LIN {X 0,Y 411.178,Z 190.084,A -85,B 0,C 180,E1 -10484.491,E2 -10484.491} C_VEL
LIN {X 0,Y 411.179,Z 190.083,A -85,B 0,C 180,E1 -10488.195,E2 -10488.195} C_VEL
LIN {X 0,Y 411.222,Z 190.077,A -85,B 0,C 180,E1 -10490.776,E2 -10490.776} C_VEL
LIN {X 0,Y 411.215,Z 190.215,A -85,B 0,C 180,E1 -10492.954,E2 -10492.954} C_VEL
LIN {X 0,Y 412.247,Z 195.412,A -85,B 0,C 180,E1 -10495.765,E2 -10495.765} C_VEL
LIN {X 0,Y 413.023,Z 200.45,A -85,B 0,C 180,E1 -10498.299,E2 -10498.299} C_VEL
LIN {X 0,Y 412.701,Z 205.041,A -85,B 0,C 180,E1 -10500.406,E2 -10500.406} C_VEL
LIN {X 0,Y 411.967,Z 212.522,A -85,B 0,C 180,E1 -10503.67,E2 -10503.67} C_VEL
LIN {X 0,Y 411.402,Z 220.138,A -85,B 0,C 180,E1 -10506.864,E2 -10506.864} C_VEL
LIN {X 0,Y 410.884,Z 229.318,A -85,B 0,C 180,E1 -10510.596,E2 -10510.596} C_VEL
LIN {X 0,Y 410.423,Z 239.572,A -85,B 0,C 180,E1 -10514.608,E2 -10514.608} C_VEL
LIN {X 0,Y 410.27,Z 243.414,A -85,B 0,C 180,E1 -10516.093,E2 -10516.093} C_VEL
LIN {X 0,Y 411.974,Z 256.351,A -85,B 0,C 180,E1 -10516.662,E2 -10516.662} C_VEL
LIN {X 0,Y 412.639,Z 265.647,A -85,B 0,C 180,E1 -10517.208,E2 -10517.208} C_VEL
LIN {X 0,Y 412.418,Z 274.261,A -85,B 0,C 180,E1 -10517.826,E2 -10517.826} C_VEL
LIN {X 0,Y 411.868,Z 282.527,A -85,B 0,C 180,E1 -10518.559,E2 -10518.559} C_VEL
LIN {X 0,Y 411.453,Z 290.378,A -85,B 0,C 180,E1 -10519.419,E2 -10519.419} C_VEL
LIN {X 0,Y 410.999,Z 297.735,A -85,B 0,C 180,E1 -10520.403,E2 -10520.403} C_VEL
LIN {X 0,Y 410.581,Z 305.203,A -85,B 0,C 180,E1 -10521.634,E2 -10521.634} C_VEL
LIN {X 0,Y 410.3,Z 311.045,A -85,B 0,C 180,E1 -10522.866,E2 -10522.866} C_VEL
LIN {X 0,Y 410.073,Z 315.663,A -85,B 0,C 180,E1 -10524.098,E2 -10524.098} C_VEL
LIN {X 0,Y 410.069,Z 318.666,A -85,B 0,C 180,E1 -10525.084,E2 -10525.084} C_VEL
LIN {X 0,Y 409.971,Z 321.016,A -85,B 0,C 180,E1 -10526.068,E2 -10526.068} C_VEL
LIN {X 0,Y 409.986,Z 322.747,A -85,B 0,C 180,E1 -10527.052,E2 -10527.052} C_VEL
LIN {X 0,Y 410.02,Z 323.966,A -85,B 0,C 180,E1 -10528.036,E2 -10528.036} C_VEL
LIN {X 0,Y 409.979,Z 324.696,A -85,B 0,C 180,E1 -10529.018,E2 -10529.018} C_VEL
LIN {X 0,Y 409.975,Z 324.952,A -85,B 0,C 180,E1 -10530,E2 -10530} C_VEL
LIN {X 0,Y 409.979,Z 324.652,A -85,B 0,C 180,E1 -10530.982,E2 -10530.982} C_VEL
LIN {X 0,Y 410.022,Z 323.785,A -85,B 0,C 180,E1 -10531.965,E2 -10531.965} C_VEL
LIN {X 0,Y 410.003,Z 322.422,A -85,B 0,C 180,E1 -10532.948,E2 -10532.948} C_VEL
LIN {X 0,Y 410.019,Z 319.386,A -85,B 0,C 180,E1 -10534.424,E2 -10534.424} C_VEL
LIN {X 0,Y 410.058,Z 315.019,A -85,B 0,C 180,E1 -10535.903,E2 -10535.903} C_VEL
LIN {X 0,Y 410.301,Z 310.119,A -85,B 0,C 180,E1 -10537.134,E2 -10537.134} C_VEL
LIN {X 0,Y 410.535,Z 303.893,A -85,B 0,C 180,E1 -10538.367,E2 -10538.367} C_VEL
LIN {X 0,Y 410.85,Z 297.806,A -85,B 0,C 180,E1 -10539.353,E2 -10539.353} C_VEL
LIN {X 0,Y 411.256,Z 290.392,A -85,B 0,C 180,E1 -10540.337,E2 -10540.337} C_VEL
LIN {X 0,Y 411.655,Z 282.441,A -85,B 0,C 180,E1 -10541.198,E2 -10541.198} C_VEL
LIN {X 0,Y 412.183,Z 272.525,A -85,B 0,C 180,E1 -10542.056,E2 -10542.056} C_VEL
LIN {X 0,Y 412.205,Z 264.215,A -85,B 0,C 180,E1 -10542.618,E2 -10542.618} C_VEL
LIN {X 0,Y 411.237,Z 253.02,A -85,B 0,C 180,E1 -10543.199,E2 -10543.199} C_VEL
LIN {X 0,Y 410.259,Z 244.088,A -85,B 0,C 180,E1 -10543.564,E2 -10543.564} C_VEL
LIN {X 0,Y 410.555,Z 235.397,A -85,B 0,C 180,E1 -10546.919,E2 -10546.919} C_VEL
LIN {X 0,Y 410.898,Z 227.517,A -85,B 0,C 180,E1 -10550.004,E2 -10550.004} C_VEL
LIN {X 0,Y 411.352,Z 219.645,A -85,B 0,C 180,E1 -10553.139,E2 -10553.139} C_VEL
LIN {X 0,Y 411.895,Z 211.789,A -85,B 0,C 180,E1 -10556.336,E2 -10556.336} C_VEL
LIN {X 0,Y 412.58,Z 203.75,A -85,B 0,C 180,E1 -10559.686,E2 -10559.686} C_VEL
LIN {X 0,Y 412.789,Z 199.19,A -85,B 0,C 180,E1 -10561.648,E2 -10561.648} C_VEL
LIN {X 0,Y 411.614,Z 192.001,A -85,B 0,C 180,E1 -10564.958,E2 -10564.958} C_VEL
LIN {X 0,Y 411.229,Z 190.075,A -85,B 0,C 180,E1 -10565.978,E2 -10565.978} C_VEL
LIN {X 0,Y 411.215,Z 190.075,A -85,B 0,C 180,E1 -10569.727,E2 -10569.727} C_VEL
LIN {X 0,Y 411.177,Z 190.079,A -85,B 0,C 180,E1 -10573.134,E2 -10573.134} C_VEL
LIN {X 0,Y 411.171,Z 190.081,A -85,B 0,C 180,E1 -10575.881,E2 -10575.881} C_VEL
LIN {X 0,Y 411.162,Z 190.083,A -85,B 0,C 180,E1 -10578.773,E2 -10578.773} C_VEL
LIN {X 0,Y 411.191,Z 190.081,A -85,B 0,C 180,E1 -10582.025,E2 -10582.025} C_VEL
LIN {X 0,Y 411.21,Z 190.076,A -85,B 0,C 180,E1 -10585.666,E2 -10585.666} C_VEL
LIN {X 0,Y 411.194,Z 190.076,A -85,B 0,C 180,E1 -10589.152,E2 -10589.152} C_VEL
LIN {X 0,Y 411.263,Z 190.068,A -85,B 0,C 180,E1 -10592.522,E2 -10592.522} C_VEL
LIN {X 0,Y 411.224,Z 190.076,A -85,B 0,C 180,E1 -10595.784,E2 -10595.784} C_VEL
LIN {X 0,Y 411.201,Z 190.076,A -85,B 0,C 180,E1 -10598.965,E2 -10598.965} C_VEL
LIN {X 0,Y 411.255,Z 190.071,A -85,B 0,C 180,E1 -10602.084,E2 -10602.084} C_VEL
LIN {X 0,Y 411.265,Z 190.07,A -85,B 0,C 180,E1 -10605.147,E2 -10605.147} C_VEL
LIN {X 0,Y 411.287,Z 190.066,A -85,B 0,C 180,E1 -10608.167,E2 -10608.167} C_VEL
LIN {X 0,Y 411.442,Z 190.046,A -85,B 0,C 180,E1 -10612.191,E2 -10612.191} C_VEL
LIN {X 0,Y 411.47,Z 190.042,A -85,B 0,C 180,E1 -10614.117,E2 -10614.117} C_VEL
LIN {X 0,Y 411.514,Z 190.036,A -85,B 0,C 180,E1 -10618.042,E2 -10618.042} C_VEL
LIN {X 0,Y 411.642,Z 190.021,A -85,B 0,C 180,E1 -10619.999,E2 -10619.999} C_VEL
LIN {X 0,Y 411.46,Z 190.047,A -85,B 0,C 180,E1 -10622.936,E2 -10622.936} C_VEL
LIN {X 0,Y 411.435,Z 190.048,A -85,B 0,C 180,E1 -10626.651,E2 -10626.651} C_VEL
LIN {X 0,Y 411.321,Z 190.064,A -85,B 0,C 180,E1 -10628.845,E2 -10628.845} C_VEL
LIN {X 0,Y 411.285,Z 190.065,A -85,B 0,C 180,E1 -10631.832,E2 -10631.832} C_VEL
LIN {X 0,Y 411.262,Z 190.071,A -85,B 0,C 180,E1 -10634.852,E2 -10634.852} C_VEL
LIN {X 0,Y 411.247,Z 190.07,A -85,B 0,C 180,E1 -10637.914,E2 -10637.914} C_VEL
LIN {X 0,Y 411.197,Z 190.078,A -85,B 0,C 180,E1 -10641.033,E2 -10641.033} C_VEL
LIN {X 0,Y 411.219,Z 190.075,A -85,B 0,C 180,E1 -10644.215,E2 -10644.215} C_VEL
LIN {X 0,Y 411.258,Z 190.068,A -85,B 0,C 180,E1 -10647.476,E2 -10647.476} C_VEL
LIN {X 0,Y 411.188,Z 190.079,A -85,B 0,C 180,E1 -10650.846,E2 -10650.846} C_VEL
LIN {X 0,Y 411.204,Z 190.079,A -85,B 0,C 180,E1 -10654.332,E2 -10654.332} C_VEL
LIN {X 0,Y 411.196,Z 190.079,A -85,B 0,C 180,E1 -10657.972,E2 -10657.972} C_VEL
LIN {X 0,Y 411.16,Z 190.081,A -85,B 0,C 180,E1 -10661.227,E2 -10661.227} C_VEL
LIN {X 0,Y 411.171,Z 190.081,A -85,B 0,C 180,E1 -10664.489,E2 -10664.489} C_VEL
LIN {X 0,Y 411.172,Z 190.082,A -85,B 0,C 180,E1 -10668.194,E2 -10668.194} C_VEL
LIN {X 0,Y 411.213,Z 190.074,A -85,B 0,C 180,E1 -10670.775,E2 -10670.775} C_VEL
LIN {X 0,Y 411.194,Z 190.077,A -85,B 0,C 180,E1 -10674.47,E2 -10674.47} C_VEL
LIN {X 0,Y 411.201,Z 190.076,A -85,B 0,C 180,E1 -10676.872,E2 -10676.872} C_VEL
LIN {X 0,Y 411.234,Z 190.071,A -85,B 0,C 180,E1 -10680.641,E2 -10680.641} C_VEL
LIN {X 0,Y 411.231,Z 190.075,A -85,B 0,C 180,E1 -10683.618,E2 -10683.618} C_VEL
LIN {X 0,Y 411.196,Z 190.078,A -85,B 0,C 180,E1 -10686.852,E2 -10686.852} C_VEL
LIN {X 0,Y 411.207,Z 190.076,A -85,B 0,C 180,E1 -10690.05,E2 -10690.05} C_VEL
LIN {X 0,Y 411.255,Z 190.073,A -85,B 0,C 180,E1 -10693.131,E2 -10693.131} C_VEL
LIN {X 0,Y 411.306,Z 190.066,A -85,B 0,C 180,E1 -10696.89,E2 -10696.89} C_VEL
LIN {X 0,Y 411.3,Z 190.062,A -85,B 0,C 180,E1 -10700.161,E2 -10700.161} C_VEL
LIN {X 0,Y 411.452,Z 190.048,A -85,B 0,C 180,E1 -10703.133,E2 -10703.133} C_VEL
LIN {X 0,Y 411.302,Z 190.066,A -85,B 0,C 180,E1 -10705.099,E2 -10705.099} C_VEL
LIN {X 0,Y 411.502,Z 190.038,A -85,B 0,C 180,E1 -10708.042,E2 -10708.042} C_VEL
LIN {X 0,Y 411.632,Z 190.023,A -85,B 0,C 180,E1 -10710,E2 -10710} C_VEL
LIN {X 0,Y 411.458,Z 190.047,A -85,B 0,C 180,E1 -10712.937,E2 -10712.937} C_VEL
LIN {X 0,Y 411.452,Z 190.048,A -85,B 0,C 180,E1 -10716.867,E2 -10716.867} C_VEL
LIN {X 0,Y 411.284,Z 190.066,A -85,B 0,C 180,E1 -10719.839,E2 -10719.839} C_VEL
LIN {X 0,Y 411.183,Z 190.079,A -85,B 0,C 180,E1 -10723.036,E2 -10723.036} C_VEL
LIN {X 0,Y 410.902,Z 190.278,A -85,B 0,C 180,E1 -10725.246,E2 -10725.246} C_VEL
LIN {X 0,Y 410.713,Z 193.427,A -85,B 0,C 180,E1 -10727.532,E2 -10727.532} C_VEL
LIN {X 0,Y 410.016,Z 194.606,A -85,B 0,C 180,E1 -10728.334,E2 -10728.334} C_VEL
LIN {X 0,Y 407.098,Z 196.713,A -85,B 0,C 180,E1 -10729.629,E2 -10729.629} C_VEL
LIN {X 0,Y 404.627,Z 198.422,A -85,B 0,C 180,E1 -10730.675,E2 -10730.675} C_VEL
LIN {X 0,Y 403.552,Z 199.659,A -85,B 0,C 180,E1 -10731.487,E2 -10731.487} C_VEL
LIN {X 0,Y 403.456,Z 200.052,A -85,B 0,C 180,E1 -10731.763,E2 -10731.763} C_VEL
LIN {X 0,Y 403.355,Z 204.668,A -85,B 0,C 180,E1 -10735.04,E2 -10735.04} C_VEL
LIN {X 0,Y 403.161,Z 209.044,A -85,B 0,C 180,E1 -10738.078,E2 -10738.078} C_VEL
LIN {X 0,Y 403.076,Z 214.046,A -85,B 0,C 180,E1 -10741.539,E2 -10741.539} C_VEL
LIN {X 0,Y 403.1,Z 215.01,A -85,B 0,C 180,E1 -10742.198,E2 -10742.198} C_VEL
LIN {X 0,Y 404.878,Z 226.111,A -85,B 0,C 180,E1 -10742.766,E2 -10742.766} C_VEL
LIN {X 0,Y 405.712,Z 233.225,A -85,B 0,C 180,E1 -10743.22,E2 -10743.22} C_VEL
LIN {X 0,Y 405.369,Z 241.394,A -85,B 0,C 180,E1 -10743.831,E2 -10743.831} C_VEL
LIN {X 0,Y 404.943,Z 249.974,A -85,B 0,C 180,E1 -10744.638,E2 -10744.638} C_VEL
LIN {X 0,Y 404.499,Z 258.989,A -85,B 0,C 180,E1 -10745.719,E2 -10745.719} C_VEL
LIN {X 0,Y 403.997,Z 266.31,A -85,B 0,C 180,E1 -10746.851,E2 -10746.851} C_VEL
LIN {X 0,Y 403.727,Z 272.109,A -85,B 0,C 180,E1 -10747.965,E2 -10747.965} C_VEL
LIN {X 0,Y 403.404,Z 276.9,A -85,B 0,C 180,E1 -10749.106,E2 -10749.106} C_VEL
LIN {X 0,Y 403.171,Z 280.422,A -85,B 0,C 180,E1 -10750.164,E2 -10750.164} C_VEL
LIN {X 0,Y 403.026,Z 283.832,A -85,B 0,C 180,E1 -10751.502,E2 -10751.502} C_VEL
LIN {X 0,Y 402.89,Z 286.206,A -85,B 0,C 180,E1 -10752.893,E2 -10752.893} C_VEL
LIN {X 0,Y 402.798,Z 287.454,A -85,B 0,C 180,E1 -10754.329,E2 -10754.329} C_VEL
LIN {X 0,Y 402.815,Z 287.615,A -85,B 0,C 180,E1 -10755.744,E2 -10755.744} C_VEL
LIN {X 0,Y 402.897,Z 286.745,A -85,B 0,C 180,E1 -10757.134,E2 -10757.134} C_VEL
LIN {X 0,Y 403.084,Z 284.77,A -85,B 0,C 180,E1 -10758.567,E2 -10758.567} C_VEL
LIN {X 0,Y 403.33,Z 281.4,A -85,B 0,C 180,E1 -10760.058,E2 -10760.058} C_VEL
LIN {X 0,Y 403.701,Z 276.409,A -85,B 0,C 180,E1 -10761.573,E2 -10761.573} C_VEL
LIN {X 0,Y 404.085,Z 270.92,A -85,B 0,C 180,E1 -10762.846,E2 -10762.846} C_VEL
LIN {X 0,Y 404.499,Z 264.45,A -85,B 0,C 180,E1 -10764.027,E2 -10764.027} C_VEL
LIN {X 0,Y 405.021,Z 257.168,A -85,B 0,C 180,E1 -10765.068,E2 -10765.068} C_VEL
LIN {X 0,Y 405.573,Z 248.818,A -85,B 0,C 180,E1 -10766.026,E2 -10766.026} C_VEL
LIN {X 0,Y 405.98,Z 240.315,A -85,B 0,C 180,E1 -10766.808,E2 -10766.808} C_VEL
LIN {X 0,Y 406.382,Z 233.7,A -85,B 0,C 180,E1 -10767.288,E2 -10767.288} C_VEL
LIN {X 0,Y 405.299,Z 226.36,A -85,B 0,C 180,E1 -10767.779,E2 -10767.779} C_VEL
LIN {X 0,Y 403.19,Z 215.872,A -85,B 0,C 180,E1 -10768.362,E2 -10768.362} C_VEL
LIN {X 0,Y 403.325,Z 212.478,A -85,B 0,C 180,E1 -10770.798,E2 -10770.798} C_VEL
LIN {X 0,Y 403.422,Z 207.853,A -85,B 0,C 180,E1 -10774.183,E2 -10774.183} C_VEL
LIN {X 0,Y 403.619,Z 203.416,A -85,B 0,C 180,E1 -10777.477,E2 -10777.477} C_VEL
LIN {X 0,Y 403.827,Z 199.168,A -85,B 0,C 180,E1 -10780.692,E2 -10780.692} C_VEL
LIN {X 0,Y 404.022,Z 195.141,A -85,B 0,C 180,E1 -10783.841,E2 -10783.841} C_VEL
LIN {X 0,Y 404.185,Z 191.247,A -85,B 0,C 180,E1 -10786.937,E2 -10786.937} C_VEL
LIN {X 0,Y 404.24,Z 190.947,A -85,B 0,C 180,E1 -10788.976,E2 -10788.976} C_VEL
LIN {X 0,Y 404.434,Z 190.926,A -85,B 0,C 180,E1 -10792.101,E2 -10792.101} C_VEL
LIN {X 0,Y 404.424,Z 190.928,A -85,B 0,C 180,E1 -10794.016,E2 -10794.016} C_VEL
LIN {X 0,Y 404.482,Z 190.917,A -85,B 0,C 180,E1 -10798.009,E2 -10798.009} C_VEL
LIN {X 0,Y 404.613,Z 190.899,A -85,B 0,C 180,E1 -10800.001,E2 -10800.001} C_VEL
LIN {X 0,Y 404.417,Z 190.921,A -85,B 0,C 180,E1 -10802.989,E2 -10802.989} C_VEL
LIN {X 0,Y 404.42,Z 190.924,A -85,B 0,C 180,E1 -10805.986,E2 -10805.986} C_VEL
LIN {X 0,Y 404.268,Z 190.941,A -85,B 0,C 180,E1 -10809.002,E2 -10809.002} C_VEL
LIN {X 0,Y 404.259,Z 190.943,A -85,B 0,C 180,E1 -10812.042,E2 -10812.042} C_VEL
LIN {X 0,Y 404.209,Z 190.95,A -85,B 0,C 180,E1 -10815.119,E2 -10815.119} C_VEL
LIN {X 0,Y 404.213,Z 190.949,A -85,B 0,C 180,E1 -10818.239,E2 -10818.239} C_VEL
LIN {X 0,Y 404.141,Z 190.957,A -85,B 0,C 180,E1 -10821.42,E2 -10821.42} C_VEL
LIN {X 0,Y 404.179,Z 190.952,A -85,B 0,C 180,E1 -10824.666,E2 -10824.666} C_VEL
LIN {X 0,Y 404.198,Z 190.951,A -85,B 0,C 180,E1 -10828,E2 -10828} C_VEL
LIN {X 0,Y 404.142,Z 190.957,A -85,B 0,C 180,E1 -10831.558,E2 -10831.558} C_VEL
LIN {X 0,Y 404.187,Z 190.951,A -85,B 0,C 180,E1 -10835.017,E2 -10835.017} C_VEL
LIN {X 0,Y 404.154,Z 190.956,A -85,B 0,C 180,E1 -10838.758,E2 -10838.758} C_VEL
LIN {X 0,Y 404.125,Z 190.962,A -85,B 0,C 180,E1 -10841.6,E2 -10841.6} C_VEL
LIN {X 0,Y 404.147,Z 190.96,A -85,B 0,C 180,E1 -10844.522,E2 -10844.522} C_VEL
LIN {X 0,Y 404.139,Z 190.961,A -85,B 0,C 180,E1 -10847.296,E2 -10847.296} C_VEL
LIN {X 0,Y 404.171,Z 190.955,A -85,B 0,C 180,E1 -10849.956,E2 -10849.956} C_VEL
LIN {X 0,Y 404.18,Z 191.105,A -85,B 0,C 180,E1 -10852.605,E2 -10852.605} C_VEL
LIN {X 0,Y 405.256,Z 196.666,A -85,B 0,C 180,E1 -10855.694,E2 -10855.694} C_VEL
LIN {X 0,Y 406.016,Z 201.16,A -85,B 0,C 180,E1 -10858.014,E2 -10858.014} C_VEL
LIN {X 0,Y 405.797,Z 205.37,A -85,B 0,C 180,E1 -10859.992,E2 -10859.992} C_VEL
LIN {X 0,Y 405.048,Z 212.468,A -85,B 0,C 180,E1 -10863.184,E2 -10863.184} C_VEL
LIN {X 0,Y 404.44,Z 220.013,A -85,B 0,C 180,E1 -10866.442,E2 -10866.442} C_VEL
LIN {X 0,Y 403.889,Z 228.575,A -85,B 0,C 180,E1 -10869.993,E2 -10869.993} C_VEL
LIN {X 0,Y 403.425,Z 238.066,A -85,B 0,C 180,E1 -10873.816,E2 -10873.816} C_VEL
LIN {X 0,Y 403.244,Z 243.125,A -85,B 0,C 180,E1 -10875.813,E2 -10875.813} C_VEL
LIN {X 0,Y 404.942,Z 255.894,A -85,B 0,C 180,E1 -10876.389,E2 -10876.389} C_VEL
LIN {X 0,Y 405.657,Z 265.712,A -85,B 0,C 180,E1 -10876.984,E2 -10876.984} C_VEL
LIN {X 0,Y 405.466,Z 274.229,A -85,B 0,C 180,E1 -10877.614,E2 -10877.614} C_VEL
LIN {X 0,Y 404.922,Z 282.429,A -85,B 0,C 180,E1 -10878.36,E2 -10878.36} C_VEL
LIN {X 0,Y 404.471,Z 290.228,A -85,B 0,C 180,E1 -10879.235,E2 -10879.235} C_VEL
LIN {X 0,Y 403.98,Z 297.545,A -85,B 0,C 180,E1 -10880.234,E2 -10880.234} C_VEL
LIN {X 0,Y 403.537,Z 304.98,A -85,B 0,C 180,E1 -10881.487,E2 -10881.487} C_VEL
LIN {X 0,Y 403.235,Z 310.795,A -85,B 0,C 180,E1 -10882.741,E2 -10882.741} C_VEL
LIN {X 0,Y 402.987,Z 315.398,A -85,B 0,C 180,E1 -10883.994,E2 -10883.994} C_VEL
LIN {X 0,Y 402.949,Z 319.567,A -85,B 0,C 180,E1 -10885.499,E2 -10885.499} C_VEL
LIN {X 0,Y 402.885,Z 322.456,A -85,B 0,C 180,E1 -10887,E2 -10887} C_VEL
LIN {X 0,Y 402.949,Z 323.662,A -85,B 0,C 180,E1 -10888.001,E2 -10888.001} C_VEL
LIN {X 0,Y 402.904,Z 324.376,A -85,B 0,C 180,E1 -10889.001,E2 -10889.001} C_VEL
LIN {X 0,Y 402.897,Z 324.617,A -85,B 0,C 180,E1 -10890,E2 -10890} C_VEL
LIN {X 0,Y 402.904,Z 324.315,A -85,B 0,C 180,E1 -10891,E2 -10891} C_VEL
LIN {X 0,Y 402.951,Z 323.434,A -85,B 0,C 180,E1 -10891.999,E2 -10891.999} C_VEL
LIN {X 0,Y 402.903,Z 322.051,A -85,B 0,C 180,E1 -10893,E2 -10893} C_VEL
LIN {X 0,Y 402.949,Z 318.997,A -85,B 0,C 180,E1 -10894.502,E2 -10894.502} C_VEL
LIN {X 0,Y 402.987,Z 314.591,A -85,B 0,C 180,E1 -10896.007,E2 -10896.007} C_VEL
LIN {X 0,Y 403.236,Z 309.652,A -85,B 0,C 180,E1 -10897.26,E2 -10897.26} C_VEL
LIN {X 0,Y 403.496,Z 303.395,A -85,B 0,C 180,E1 -10898.514,E2 -10898.514} C_VEL
LIN {X 0,Y 403.802,Z 297.268,A -85,B 0,C 180,E1 -10899.517,E2 -10899.517} C_VEL
LIN {X 0,Y 404.187,Z 290.833,A -85,B 0,C 180,E1 -10900.393,E2 -10900.393} C_VEL
LIN {X 0,Y 404.501,Z 284.26,A -85,B 0,C 180,E1 -10901.145,E2 -10901.145} C_VEL
LIN {X 0,Y 404.992,Z 276.317,A -85,B 0,C 180,E1 -10901.892,E2 -10901.892} C_VEL
LIN {X 0,Y 405.311,Z 268.134,A -85,B 0,C 180,E1 -10902.517,E2 -10902.517} C_VEL
LIN {X 0,Y 404.813,Z 259.719,A -85,B 0,C 180,E1 -10903.044,E2 -10903.044} C_VEL
LIN {X 0,Y 403.871,Z 250.187,A -85,B 0,C 180,E1 -10903.507,E2 -10903.507} C_VEL
LIN {X 0,Y 403.178,Z 243.814,A -85,B 0,C 180,E1 -10903.772,E2 -10903.772} C_VEL
LIN {X 0,Y 403.497,Z 235.076,A -85,B 0,C 180,E1 -10907.224,E2 -10907.224} C_VEL
LIN {X 0,Y 403.894,Z 227.242,A -85,B 0,C 180,E1 -10910.366,E2 -10910.366} C_VEL
LIN {X 0,Y 404.441,Z 218.064,A -85,B 0,C 180,E1 -10914.102,E2 -10914.102} C_VEL
LIN {X 0,Y 405.052,Z 210.38,A -85,B 0,C 180,E1 -10917.306,E2 -10917.306} C_VEL
LIN {X 0,Y 405.77,Z 202.419,A -85,B 0,C 180,E1 -10920.727,E2 -10920.727} C_VEL
LIN {X 0,Y 405.501,Z 198.472,A -85,B 0,C 180,E1 -10922.499,E2 -10922.499} C_VEL
LIN {X 0,Y 404.344,Z 191.755,A -85,B 0,C 180,E1 -10925.695,E2 -10925.695} C_VEL
LIN {X 0,Y 404.182,Z 190.954,A -85,B 0,C 180,E1 -10926.109,E2 -10926.109} C_VEL
LIN {X 0,Y 404.156,Z 190.957,A -85,B 0,C 180,E1 -10928.757,E2 -10928.757} C_VEL
LIN {X 0,Y 404.126,Z 190.957,A -85,B 0,C 180,E1 -10931.6,E2 -10931.6} C_VEL
LIN {X 0,Y 404.149,Z 190.957,A -85,B 0,C 180,E1 -10934.522,E2 -10934.522} C_VEL
LIN {X 0,Y 404.136,Z 190.955,A -85,B 0,C 180,E1 -10937.295,E2 -10937.295} C_VEL
LIN {X 0,Y 404.136,Z 190.958,A -85,B 0,C 180,E1 -10939.951,E2 -10939.951} C_VEL
LIN {X 0,Y 404.139,Z 190.955,A -85,B 0,C 180,E1 -10943.125,E2 -10943.125} C_VEL
LIN {X 0,Y 404.149,Z 190.957,A -85,B 0,C 180,E1 -10946.188,E2 -10946.188} C_VEL
LIN {X 0,Y 404.15,Z 190.957,A -85,B 0,C 180,E1 -10949.715,E2 -10949.715} C_VEL
LIN {X 0,Y 404.199,Z 190.947,A -85,B 0,C 180,E1 -10953.123,E2 -10953.123} C_VEL
LIN {X 0,Y 404.178,Z 190.952,A -85,B 0,C 180,E1 -10955.334,E2 -10955.334} C_VEL
LIN {X 0,Y 404.143,Z 190.955,A -85,B 0,C 180,E1 -10958.58,E2 -10958.58} C_VEL
LIN {X 0,Y 404.213,Z 190.949,A -85,B 0,C 180,E1 -10961.761,E2 -10961.761} C_VEL
LIN {X 0,Y 404.211,Z 190.947,A -85,B 0,C 180,E1 -10964.881,E2 -10964.881} C_VEL
LIN {X 0,Y 404.26,Z 190.942,A -85,B 0,C 180,E1 -10967.958,E2 -10967.958} C_VEL
LIN {X 0,Y 404.27,Z 190.94,A -85,B 0,C 180,E1 -10970.998,E2 -10970.998} C_VEL
LIN {X 0,Y 404.417,Z 190.921,A -85,B 0,C 180,E1 -10974.014,E2 -10974.014} C_VEL
LIN {X 0,Y 404.483,Z 190.912,A -85,B 0,C 180,E1 -10978.008,E2 -10978.008} C_VEL
LIN {X 0,Y 404.611,Z 190.897,A -85,B 0,C 180,E1 -10979.999,E2 -10979.999} C_VEL
LIN {X 0,Y 404.418,Z 190.924,A -85,B 0,C 180,E1 -10982.988,E2 -10982.988} C_VEL
LIN {X 0,Y 404.384,Z 190.925,A -85,B 0,C 180,E1 -10986.65,E2 -10986.65} C_VEL
LIN {X 0,Y 404.259,Z 190.94,A -85,B 0,C 180,E1 -10990.011,E2 -10990.011} C_VEL
LIN {X 0,Y 404.268,Z 190.941,A -85,B 0,C 180,E1 -10993.21,E2 -10993.21} C_VEL
LIN {X 0,Y 404.217,Z 190.948,A -85,B 0,C 180,E1 -10997.006,E2 -10997.006} C_VEL
LIN {X 0,Y 404.164,Z 190.954,A -85,B 0,C 180,E1 -11000.35,E2 -11000.35} C_VEL
LIN {X 0,Y 404.163,Z 190.952,A -85,B 0,C 180,E1 -11003.574,E2 -11003.574} C_VEL
LIN {X 0,Y 404.182,Z 190.95,A -85,B 0,C 180,E1 -11005.765,E2 -11005.765} C_VEL
LIN {X 0,Y 404.195,Z 190.95,A -85,B 0,C 180,E1 -11007.998,E2 -11007.998} C_VEL
LIN {X 0,Y 404.138,Z 190.955,A -85,B 0,C 180,E1 -11011.557,E2 -11011.557} C_VEL
LIN {X 0,Y 404.183,Z 190.949,A -85,B 0,C 180,E1 -11015.015,E2 -11015.015} C_VEL
LIN {X 0,Y 404.153,Z 190.953,A -85,B 0,C 180,E1 -11018.756,E2 -11018.756} C_VEL
LIN {X 0,Y 404.119,Z 190.96,A -85,B 0,C 180,E1 -11021.599,E2 -11021.599} C_VEL
LIN {X 0,Y 404.141,Z 190.957,A -85,B 0,C 180,E1 -11024.521,E2 -11024.521} C_VEL
LIN {X 0,Y 404.132,Z 190.956,A -85,B 0,C 180,E1 -11027.295,E2 -11027.295} C_VEL
LIN {X 0,Y 404.164,Z 190.956,A -85,B 0,C 180,E1 -11029.954,E2 -11029.954} C_VEL
LIN {X 0,Y 404.134,Z 190.957,A -85,B 0,C 180,E1 -11033.123,E2 -11033.123} C_VEL
LIN {X 0,Y 404.139,Z 190.957,A -85,B 0,C 180,E1 -11036.187,E2 -11036.187} C_VEL
LIN {X 0,Y 404.147,Z 190.957,A -85,B 0,C 180,E1 -11039.715,E2 -11039.715} C_VEL
LIN {X 0,Y 404.188,Z 190.952,A -85,B 0,C 180,E1 -11043.122,E2 -11043.122} C_VEL
LIN {X 0,Y 404.17,Z 190.955,A -85,B 0,C 180,E1 -11045.334,E2 -11045.334} C_VEL
LIN {X 0,Y 404.131,Z 190.956,A -85,B 0,C 180,E1 -11048.58,E2 -11048.58} C_VEL
LIN {X 0,Y 404.202,Z 190.948,A -85,B 0,C 180,E1 -11051.761,E2 -11051.761} C_VEL
LIN {X 0,Y 404.201,Z 190.95,A -85,B 0,C 180,E1 -11054.882,E2 -11054.882} C_VEL
LIN {X 0,Y 404.263,Z 190.94,A -85,B 0,C 180,E1 -11057.958,E2 -11057.958} C_VEL
LIN {X 0,Y 404.425,Z 190.92,A -85,B 0,C 180,E1 -11062.099,E2 -11062.099} C_VEL
LIN {X 0,Y 404.415,Z 190.92,A -85,B 0,C 180,E1 -11064.015,E2 -11064.015} C_VEL
LIN {X 0,Y 404.471,Z 190.913,A -85,B 0,C 180,E1 -11068.008,E2 -11068.008} C_VEL
LIN {X 0,Y 404.602,Z 190.898,A -85,B 0,C 180,E1 -11070,E2 -11070} C_VEL
LIN {X 0,Y 404.414,Z 190.924,A -85,B 0,C 180,E1 -11072.988,E2 -11072.988} C_VEL
LIN {X 0,Y 404.403,Z 190.925,A -85,B 0,C 180,E1 -11076.987,E2 -11076.987} C_VEL
LIN {X 0,Y 404.248,Z 190.944,A -85,B 0,C 180,E1 -11080.012,E2 -11080.012} C_VEL
LIN {X 0,Y 404.14,Z 190.956,A -85,B 0,C 180,E1 -11083.14,E2 -11083.14} C_VEL
LIN {X 0,Y 403.849,Z 191.131,A -85,B 0,C 180,E1 -11085.261,E2 -11085.261} C_VEL
LIN {X 0,Y 403.624,Z 195.224,A -85,B 0,C 180,E1 -11088.265,E2 -11088.265} C_VEL
LIN {X 0,Y 403.478,Z 199.623,A -85,B 0,C 180,E1 -11091.456,E2 -11091.456} C_VEL
LIN {X 0,Y 403.456,Z 200.052,A -85,B 0,C 180,E1 -11091.763,E2 -11091.763} C_VEL
LIN {X 0,Y 402.754,Z 201.264,A -85,B 0,C 180,E1 -11092.577,E2 -11092.577} C_VEL
LIN {X 0,Y 399.832,Z 203.404,A -85,B 0,C 180,E1 -11093.894,E2 -11093.894} C_VEL
LIN {X 0,Y 397.365,Z 205.131,A -85,B 0,C 180,E1 -11094.957,E2 -11094.957} C_VEL
LIN {X 0,Y 396.296,Z 206.387,A -85,B 0,C 180,E1 -11095.782,E2 -11095.782} C_VEL
LIN {X 0,Y 396.203,Z 206.785,A -85,B 0,C 180,E1 -11096.063,E2 -11096.063} C_VEL
LIN {X 0,Y 396.05,Z 211.819,A -85,B 0,C 180,E1 -11099.6,E2 -11099.6} C_VEL
LIN {X 0,Y 396.023,Z 215.304,A -85,B 0,C 180,E1 -11102.007,E2 -11102.007} C_VEL
LIN {X 0,Y 397.743,Z 225.737,A -85,B 0,C 180,E1 -11102.535,E2 -11102.535} C_VEL
LIN {X 0,Y 398.74,Z 233.607,A -85,B 0,C 180,E1 -11103.044,E2 -11103.044} C_VEL
LIN {X 0,Y 398.36,Z 242.472,A -85,B 0,C 180,E1 -11103.727,E2 -11103.727} C_VEL
LIN {X 0,Y 397.835,Z 252.576,A -85,B 0,C 180,E1 -11104.73,E2 -11104.73} C_VEL
LIN {X 0,Y 397.283,Z 261.257,A -85,B 0,C 180,E1 -11105.873,E2 -11105.873} C_VEL
LIN {X 0,Y 396.971,Z 266.379,A -85,B 0,C 180,E1 -11106.692,E2 -11106.692} C_VEL
LIN {X 0,Y 396.722,Z 271.665,A -85,B 0,C 180,E1 -11107.706,E2 -11107.706} C_VEL
LIN {X 0,Y 396.442,Z 276.105,A -85,B 0,C 180,E1 -11108.74,E2 -11108.74} C_VEL
LIN {X 0,Y 396.065,Z 281.238,A -85,B 0,C 180,E1 -11110.271,E2 -11110.271} C_VEL
LIN {X 0,Y 395.909,Z 284.796,A -85,B 0,C 180,E1 -11111.794,E2 -11111.794} C_VEL
LIN {X 0,Y 395.762,Z 286.925,A -85,B 0,C 180,E1 -11113.276,E2 -11113.276} C_VEL
LIN {X 0,Y 395.691,Z 287.917,A -85,B 0,C 180,E1 -11114.73,E2 -11114.73} C_VEL
LIN {X 0,Y 395.734,Z 287.841,A -85,B 0,C 180,E1 -11116.164,E2 -11116.164} C_VEL
LIN {X 0,Y 395.867,Z 286.734,A -85,B 0,C 180,E1 -11117.576,E2 -11117.576} C_VEL
LIN {X 0,Y 396.071,Z 284.56,A -85,B 0,C 180,E1 -11118.965,E2 -11118.965} C_VEL
LIN {X 0,Y 396.324,Z 281.296,A -85,B 0,C 180,E1 -11120.33,E2 -11120.33} C_VEL
LIN {X 0,Y 396.655,Z 276.923,A -85,B 0,C 180,E1 -11121.676,E2 -11121.676} C_VEL
LIN {X 0,Y 396.996,Z 272.212,A -85,B 0,C 180,E1 -11122.81,E2 -11122.81} C_VEL
LIN {X 0,Y 397.431,Z 266.123,A -85,B 0,C 180,E1 -11123.988,E2 -11123.988} C_VEL
LIN {X 0,Y 398.085,Z 257.377,A -85,B 0,C 180,E1 -11125.296,E2 -11125.296} C_VEL
LIN {X 0,Y 398.558,Z 250.876,A -85,B 0,C 180,E1 -11126.073,E2 -11126.073} C_VEL
LIN {X 0,Y 398.99,Z 242.332,A -85,B 0,C 180,E1 -11126.905,E2 -11126.905} C_VEL
LIN {X 0,Y 399.446,Z 233.952,A -85,B 0,C 180,E1 -11127.548,E2 -11127.548} C_VEL
LIN {X 0,Y 397.846,Z 224.533,A -85,B 0,C 180,E1 -11128.188,E2 -11128.188} C_VEL
LIN {X 0,Y 396.149,Z 216.171,A -85,B 0,C 180,E1 -11128.65,E2 -11128.65} C_VEL
LIN {X 0,Y 396.303,Z 210.973,A -85,B 0,C 180,E1 -11132.461,E2 -11132.461} C_VEL
LIN {X 0,Y 396.464,Z 206.322,A -85,B 0,C 180,E1 -11135.94,E2 -11135.94} C_VEL
LIN {X 0,Y 396.671,Z 201.983,A -85,B 0,C 180,E1 -11139.248,E2 -11139.248} C_VEL
LIN {X 0,Y 396.928,Z 197.251,A -85,B 0,C 180,E1 -11142.964,E2 -11142.964} C_VEL
LIN {X 0,Y 397.077,Z 193.887,A -85,B 0,C 180,E1 -11145.654,E2 -11145.654} C_VEL
LIN {X 0,Y 397.148,Z 192.582,A -85,B 0,C 180,E1 -11146.728,E2 -11146.728} C_VEL
LIN {X 0,Y 397.152,Z 191.835,A -85,B 0,C 180,E1 -11147.741,E2 -11147.741} C_VEL
LIN {X 0,Y 397.252,Z 191.818,A -85,B 0,C 180,E1 -11150.839,E2 -11150.839} C_VEL
LIN {X 0,Y 397.365,Z 191.807,A -85,B 0,C 180,E1 -11152.889,E2 -11152.889} C_VEL
LIN {X 0,Y 397.255,Z 191.82,A -85,B 0,C 180,E1 -11154.926,E2 -11154.926} C_VEL
LIN {X 0,Y 397.451,Z 191.793,A -85,B 0,C 180,E1 -11157.974,E2 -11157.974} C_VEL
LIN {X 0,Y 397.582,Z 191.775,A -85,B 0,C 180,E1 -11160.001,E2 -11160.001} C_VEL
LIN {X 0,Y 397.377,Z 191.798,A -85,B 0,C 180,E1 -11163.042,E2 -11163.042} C_VEL
LIN {X 0,Y 397.37,Z 191.801,A -85,B 0,C 180,E1 -11166.092,E2 -11166.092} C_VEL
LIN {X 0,Y 397.238,Z 191.817,A -85,B 0,C 180,E1 -11169.163,E2 -11169.163} C_VEL
LIN {X 0,Y 397.222,Z 191.819,A -85,B 0,C 180,E1 -11172.259,E2 -11172.259} C_VEL
LIN {X 0,Y 397.182,Z 191.825,A -85,B 0,C 180,E1 -11175.393,E2 -11175.393} C_VEL
LIN {X 0,Y 397.165,Z 191.827,A -85,B 0,C 180,E1 -11178.574,E2 -11178.574} C_VEL
LIN {X 0,Y 397.099,Z 191.835,A -85,B 0,C 180,E1 -11181.819,E2 -11181.819} C_VEL
LIN {X 0,Y 397.159,Z 191.825,A -85,B 0,C 180,E1 -11185.132,E2 -11185.132} C_VEL
LIN {X 0,Y 397.164,Z 191.827,A -85,B 0,C 180,E1 -11187.777,E2 -11187.777} C_VEL
LIN {X 0,Y 397.081,Z 191.837,A -85,B 0,C 180,E1 -11190.883,E2 -11190.883} C_VEL
LIN {X 0,Y 397.128,Z 191.831,A -85,B 0,C 180,E1 -11194.494,E2 -11194.494} C_VEL
LIN {X 0,Y 397.103,Z 191.835,A -85,B 0,C 180,E1 -11198.276,E2 -11198.276} C_VEL
LIN {X 0,Y 397.091,Z 191.837,A -85,B 0,C 180,E1 -11200.909,E2 -11200.909} C_VEL
LIN {X 0,Y 397.103,Z 191.838,A -85,B 0,C 180,E1 -11203.649,E2 -11203.649} C_VEL
LIN {X 0,Y 397.104,Z 191.837,A -85,B 0,C 180,E1 -11206.521,E2 -11206.521} C_VEL
LIN {X 0,Y 397.116,Z 191.834,A -85,B 0,C 180,E1 -11210.423,E2 -11210.423} C_VEL
LIN {X 0,Y 397.121,Z 191.863,A -85,B 0,C 180,E1 -11212.149,E2 -11212.149} C_VEL
LIN {X 0,Y 398.286,Z 197.939,A -85,B 0,C 180,E1 -11215.621,E2 -11215.621} C_VEL
LIN {X 0,Y 399.029,Z 202.67,A -85,B 0,C 180,E1 -11218.104,E2 -11218.104} C_VEL
LIN {X 0,Y 398.882,Z 205.967,A -85,B 0,C 180,E1 -11219.695,E2 -11219.695} C_VEL
LIN {X 0,Y 398.102,Z 212.433,A -85,B 0,C 180,E1 -11222.678,E2 -11222.678} C_VEL
LIN {X 0,Y 397.48,Z 219.962,A -85,B 0,C 180,E1 -11226.004,E2 -11226.004} C_VEL
LIN {X 0,Y 396.836,Z 228.913,A -85,B 0,C 180,E1 -11229.824,E2 -11229.824} C_VEL
LIN {X 0,Y 396.395,Z 237.879,A -85,B 0,C 180,E1 -11233.52,E2 -11233.52} C_VEL
LIN {X 0,Y 396.152,Z 242.834,A -85,B 0,C 180,E1 -11235.521,E2 -11235.521} C_VEL
LIN {X 0,Y 397.9,Z 255.576,A -85,B 0,C 180,E1 -11236.114,E2 -11236.114} C_VEL
LIN {X 0,Y 398.667,Z 265.803,A -85,B 0,C 180,E1 -11236.752,E2 -11236.752} C_VEL
LIN {X 0,Y 398.539,Z 274.237,A -85,B 0,C 180,E1 -11237.395,E2 -11237.395} C_VEL
LIN {X 0,Y 397.967,Z 282.377,A -85,B 0,C 180,E1 -11238.153,E2 -11238.153} C_VEL
LIN {X 0,Y 397.497,Z 290.132,A -85,B 0,C 180,E1 -11239.043,E2 -11239.043} C_VEL
LIN {X 0,Y 396.866,Z 299.084,A -85,B 0,C 180,E1 -11240.315,E2 -11240.315} C_VEL
LIN {X 0,Y 396.422,Z 306.003,A -85,B 0,C 180,E1 -11241.59,E2 -11241.59} C_VEL
LIN {X 0,Y 396.117,Z 311.536,A -85,B 0,C 180,E1 -11242.866,E2 -11242.866} C_VEL
LIN {X 0,Y 395.91,Z 315.145,A -85,B 0,C 180,E1 -11243.886,E2 -11243.886} C_VEL
LIN {X 0,Y 395.879,Z 319.294,A -85,B 0,C 180,E1 -11245.418,E2 -11245.418} C_VEL
LIN {X 0,Y 395.785,Z 322.166,A -85,B 0,C 180,E1 -11246.947,E2 -11246.947} C_VEL
LIN {X 0,Y 395.86,Z 323.358,A -85,B 0,C 180,E1 -11247.965,E2 -11247.965} C_VEL
LIN {X 0,Y 395.831,Z 324.057,A -85,B 0,C 180,E1 -11248.983,E2 -11248.983} C_VEL
LIN {X 0,Y 395.822,Z 324.281,A -85,B 0,C 180,E1 -11250,E2 -11250} C_VEL
LIN {X 0,Y 395.832,Z 323.977,A -85,B 0,C 180,E1 -11251.018,E2 -11251.018} C_VEL
LIN {X 0,Y 395.863,Z 323.082,A -85,B 0,C 180,E1 -11252.035,E2 -11252.035} C_VEL
LIN {X 0,Y 395.804,Z 321.68,A -85,B 0,C 180,E1 -11253.054,E2 -11253.054} C_VEL
LIN {X 0,Y 395.879,Z 318.607,A -85,B 0,C 180,E1 -11254.582,E2 -11254.582} C_VEL
LIN {X 0,Y 395.955,Z 313.5,A -85,B 0,C 180,E1 -11256.292,E2 -11256.292} C_VEL
LIN {X 0,Y 396.169,Z 309.186,A -85,B 0,C 180,E1 -11257.39,E2 -11257.39} C_VEL
LIN {X 0,Y 396.444,Z 302.896,A -85,B 0,C 180,E1 -11258.667,E2 -11258.667} C_VEL
LIN {X 0,Y 396.776,Z 296.733,A -85,B 0,C 180,E1 -11259.688,E2 -11259.688} C_VEL
LIN {X 0,Y 397.174,Z 290.252,A -85,B 0,C 180,E1 -11260.579,E2 -11260.579} C_VEL
LIN {X 0,Y 397.536,Z 283.627,A -85,B 0,C 180,E1 -11261.343,E2 -11261.343} C_VEL
LIN {X 0,Y 398.017,Z 275.611,A -85,B 0,C 180,E1 -11262.104,E2 -11262.104} C_VEL
LIN {X 0,Y 398.288,Z 267.836,A -85,B 0,C 180,E1 -11262.706,E2 -11262.706} C_VEL
LIN {X 0,Y 397.683,Z 258.753,A -85,B 0,C 180,E1 -11263.282,E2 -11263.282} C_VEL
LIN {X 0,Y 396.607,Z 248.22,A -85,B 0,C 180,E1 -11263.789,E2 -11263.789} C_VEL
LIN {X 0,Y 396.12,Z 243.663,A -85,B 0,C 180,E1 -11263.95,E2 -11263.95} C_VEL
LIN {X 0,Y 396.463,Z 234.777,A -85,B 0,C 180,E1 -11267.539,E2 -11267.539} C_VEL
LIN {X 0,Y 396.848,Z 226.939,A -85,B 0,C 180,E1 -11270.744,E2 -11270.744} C_VEL
LIN {X 0,Y 397.373,Z 219.105,A -85,B 0,C 180,E1 -11274.003,E2 -11274.003} C_VEL
LIN {X 0,Y 398.005,Z 211.302,A -85,B 0,C 180,E1 -11277.33,E2 -11277.33} C_VEL
LIN {X 0,Y 398.758,Z 203.484,A -85,B 0,C 180,E1 -11280.739,E2 -11280.739} C_VEL
LIN {X 0,Y 398.474,Z 199.385,A -85,B 0,C 180,E1 -11282.622,E2 -11282.622} C_VEL
LIN {X 0,Y 397.377,Z 193.012,A -85,B 0,C 180,E1 -11285.707,E2 -11285.707} C_VEL
LIN {X 0,Y 397.126,Z 191.832,A -85,B 0,C 180,E1 -11286.36,E2 -11286.36} C_VEL
LIN {X 0,Y 397.117,Z 191.833,A -85,B 0,C 180,E1 -11289.577,E2 -11289.577} C_VEL
LIN {X 0,Y 397.106,Z 191.831,A -85,B 0,C 180,E1 -11293.479,E2 -11293.479} C_VEL
LIN {X 0,Y 397.105,Z 191.835,A -85,B 0,C 180,E1 -11296.521,E2 -11296.521} C_VEL
LIN {X 0,Y 397.092,Z 191.837,A -85,B 0,C 180,E1 -11300.42,E2 -11300.42} C_VEL
LIN {X 0,Y 397.101,Z 191.832,A -85,B 0,C 180,E1 -11303.005,E2 -11303.005} C_VEL
LIN {X 0,Y 397.123,Z 191.832,A -85,B 0,C 180,E1 -11306.282,E2 -11306.282} C_VEL
LIN {X 0,Y 397.11,Z 191.834,A -85,B 0,C 180,E1 -11310.135,E2 -11310.135} C_VEL
LIN {X 0,Y 397.199,Z 191.82,A -85,B 0,C 180,E1 -11312.61,E2 -11312.61} C_VEL
LIN {X 0,Y 397.133,Z 191.831,A -85,B 0,C 180,E1 -11315.981,E2 -11315.981} C_VEL
LIN {X 0,Y 397.143,Z 191.831,A -85,B 0,C 180,E1 -11319.704,E2 -11319.704} C_VEL
LIN {X 0,Y 397.187,Z 191.821,A -85,B 0,C 180,E1 -11322.844,E2 -11322.844} C_VEL
LIN {X 0,Y 397.233,Z 191.815,A -85,B 0,C 180,E1 -11326.702,E2 -11326.702} C_VEL
LIN {X 0,Y 397.22,Z 191.819,A -85,B 0,C 180,E1 -11329.808,E2 -11329.808} C_VEL
LIN {X 0,Y 397.337,Z 191.804,A -85,B 0,C 180,E1 -11332.887,E2 -11332.887} C_VEL
LIN {X 0,Y 397.254,Z 191.814,A -85,B 0,C 180,E1 -11334.924,E2 -11334.924} C_VEL
LIN {X 0,Y 397.452,Z 191.788,A -85,B 0,C 180,E1 -11337.972,E2 -11337.972} C_VEL
LIN {X 0,Y 397.58,Z 191.772,A -85,B 0,C 180,E1 -11339.999,E2 -11339.999} C_VEL
LIN {X 0,Y 397.378,Z 191.801,A -85,B 0,C 180,E1 -11343.041,E2 -11343.041} C_VEL
LIN {X 0,Y 397.334,Z 191.802,A -85,B 0,C 180,E1 -11346.646,E2 -11346.646} C_VEL
LIN {X 0,Y 397.238,Z 191.818,A -85,B 0,C 180,E1 -11349.161,E2 -11349.161} C_VEL
LIN {X 0,Y 397.221,Z 191.818,A -85,B 0,C 180,E1 -11352.257,E2 -11352.257} C_VEL
LIN {X 0,Y 397.18,Z 191.823,A -85,B 0,C 180,E1 -11355.391,E2 -11355.391} C_VEL
LIN {X 0,Y 397.159,Z 191.828,A -85,B 0,C 180,E1 -11358.572,E2 -11358.572} C_VEL
LIN {X 0,Y 397.096,Z 191.833,A -85,B 0,C 180,E1 -11361.817,E2 -11361.817} C_VEL
LIN {X 0,Y 397.152,Z 191.825,A -85,B 0,C 180,E1 -11365.511,E2 -11365.511} C_VEL
LIN {X 0,Y 397.121,Z 191.832,A -85,B 0,C 180,E1 -11368.542,E2 -11368.542} C_VEL
LIN {X 0,Y 397.077,Z 191.837,A -85,B 0,C 180,E1 -11372.07,E2 -11372.07} C_VEL
LIN {X 0,Y 397.118,Z 191.829,A -85,B 0,C 180,E1 -11375.502,E2 -11375.502} C_VEL
LIN {X 0,Y 397.128,Z 191.828,A -85,B 0,C 180,E1 -11378.86,E2 -11378.86} C_VEL
LIN {X 0,Y 397.065,Z 191.839,A -85,B 0,C 180,E1 -11382.266,E2 -11382.266} C_VEL
LIN {X 0,Y 397.082,Z 191.834,A -85,B 0,C 180,E1 -11385.068,E2 -11385.068} C_VEL
LIN {X 0,Y 397.061,Z 191.84,A -85,B 0,C 180,E1 -11388.02,E2 -11388.02} C_VEL
LIN {X 0,Y 397.126,Z 191.829,A -85,B 0,C 180,E1 -11391.137,E2 -11391.137} C_VEL
LIN {X 0,Y 397.114,Z 191.83,A -85,B 0,C 180,E1 -11394.495,E2 -11394.495} C_VEL
LIN {X 0,Y 397.074,Z 191.837,A -85,B 0,C 180,E1 -11397.928,E2 -11397.928} C_VEL
LIN {X 0,Y 397.12,Z 191.833,A -85,B 0,C 180,E1 -11401.456,E2 -11401.456} C_VEL
LIN {X 0,Y 397.145,Z 191.826,A -85,B 0,C 180,E1 -11404.487,E2 -11404.487} C_VEL
LIN {X 0,Y 397.102,Z 191.835,A -85,B 0,C 180,E1 -11407.085,E2 -11407.085} C_VEL
LIN {X 0,Y 397.14,Z 191.827,A -85,B 0,C 180,E1 -11410.352,E2 -11410.352} C_VEL
LIN {X 0,Y 397.158,Z 191.827,A -85,B 0,C 180,E1 -11413.553,E2 -11413.553} C_VEL
LIN {X 0,Y 397.22,Z 191.818,A -85,B 0,C 180,E1 -11416.702,E2 -11416.702} C_VEL
LIN {X 0,Y 397.221,Z 191.816,A -85,B 0,C 180,E1 -11419.809,E2 -11419.809} C_VEL
LIN {X 0,Y 397.355,Z 191.803,A -85,B 0,C 180,E1 -11422.888,E2 -11422.888} C_VEL
LIN {X 0,Y 397.246,Z 191.817,A -85,B 0,C 180,E1 -11424.925,E2 -11424.925} C_VEL
LIN {X 0,Y 397.44,Z 191.789,A -85,B 0,C 180,E1 -11427.973,E2 -11427.973} C_VEL
LIN {X 0,Y 397.571,Z 191.774,A -85,B 0,C 180,E1 -11430,E2 -11430} C_VEL
LIN {X 0,Y 397.373,Z 191.801,A -85,B 0,C 180,E1 -11433.041,E2 -11433.041} C_VEL
LIN {X 0,Y 397.355,Z 191.801,A -85,B 0,C 180,E1 -11437.112,E2 -11437.112} C_VEL
LIN {X 0,Y 397.207,Z 191.822,A -85,B 0,C 180,E1 -11440.191,E2 -11440.191} C_VEL
LIN {X 0,Y 397.082,Z 191.834,A -85,B 0,C 180,E1 -11443.302,E2 -11443.302} C_VEL
LIN {X 0,Y 396.817,Z 191.983,A -85,B 0,C 180,E1 -11445.275,E2 -11445.275} C_VEL
LIN {X 0,Y 396.552,Z 196.456,A -85,B 0,C 180,E1 -11448.603,E2 -11448.603} C_VEL
LIN {X 0,Y 396.387,Z 200.9,A -85,B 0,C 180,E1 -11451.859,E2 -11451.859} C_VEL
LIN {X 0,Y 396.274,Z 205.644,A -85,B 0,C 180,E1 -11455.248,E2 -11455.248} C_VEL
LIN {X 0,Y 396.203,Z 206.785,A -85,B 0,C 180,E1 -11456.063,E2 -11456.063} C_VEL
LIN {X 0,Y 395.504,Z 208.014,A -85,B 0,C 180,E1 -11456.891,E2 -11456.891} C_VEL
LIN {X 0,Y 392.571,Z 210.174,A -85,B 0,C 180,E1 -11458.231,E2 -11458.231} C_VEL
LIN {X 0,Y 390.086,Z 211.922,A -85,B 0,C 180,E1 -11459.312,E2 -11459.312} C_VEL
LIN {X 0,Y 389.008,Z 213.2,A -85,B 0,C 180,E1 -11460.152,E2 -11460.152} C_VEL
LIN {X 0,Y 388.914,Z 213.611,A -85,B 0,C 180,E1 -11460.437,E2 -11460.437} C_VEL
LIN {X 0,Y 388.925,Z 215.527,A -85,B 0,C 180,E1 -11461.786,E2 -11461.786} C_VEL
LIN {X 0,Y 390.813,Z 226.869,A -85,B 0,C 180,E1 -11462.389,E2 -11462.389} C_VEL
LIN {X 0,Y 391.742,Z 235.084,A -85,B 0,C 180,E1 -11462.944,E2 -11462.944} C_VEL
LIN {X 0,Y 391.303,Z 244.182,A -85,B 0,C 180,E1 -11463.678,E2 -11463.678} C_VEL
LIN {X 0,Y 390.785,Z 253.497,A -85,B 0,C 180,E1 -11464.654,E2 -11464.654} C_VEL
LIN {X 0,Y 390.407,Z 260.006,A -85,B 0,C 180,E1 -11465.506,E2 -11465.506} C_VEL
LIN {X 0,Y 389.979,Z 266.229,A -85,B 0,C 180,E1 -11466.492,E2 -11466.492} C_VEL
LIN {X 0,Y 389.711,Z 271.436,A -85,B 0,C 180,E1 -11467.489,E2 -11467.489} C_VEL
LIN {X 0,Y 389.345,Z 276.787,A -85,B 0,C 180,E1 -11468.758,E2 -11468.758} C_VEL
LIN {X 0,Y 389.055,Z 280.567,A -85,B 0,C 180,E1 -11469.887,E2 -11469.887} C_VEL
LIN {X 0,Y 388.866,Z 284.1,A -85,B 0,C 180,E1 -11471.274,E2 -11471.274} C_VEL
LIN {X 0,Y 388.791,Z 285.766,A -85,B 0,C 180,E1 -11472.174,E2 -11472.174} C_VEL
LIN {X 0,Y 388.645,Z 287.635,A -85,B 0,C 180,E1 -11473.671,E2 -11473.671} C_VEL
LIN {X 0,Y 388.606,Z 288.382,A -85,B 0,C 180,E1 -11475.146,E2 -11475.146} C_VEL
LIN {X 0,Y 388.676,Z 288.013,A -85,B 0,C 180,E1 -11476.6,E2 -11476.6} C_VEL
LIN {X 0,Y 388.864,Z 286.553,A -85,B 0,C 180,E1 -11478.034,E2 -11478.034} C_VEL
LIN {X 0,Y 389.067,Z 284.092,A -85,B 0,C 180,E1 -11479.438,E2 -11479.438} C_VEL
LIN {X 0,Y 389.204,Z 282.548,A -85,B 0,C 180,E1 -11480.132,E2 -11480.132} C_VEL
LIN {X 0,Y 389.548,Z 278.273,A -85,B 0,C 180,E1 -11481.552,E2 -11481.552} C_VEL
LIN {X 0,Y 389.918,Z 273.61,A -85,B 0,C 180,E1 -11482.747,E2 -11482.747} C_VEL
LIN {X 0,Y 390.345,Z 268.199,A -85,B 0,C 180,E1 -11483.862,E2 -11483.862} C_VEL
LIN {X 0,Y 390.829,Z 262.204,A -85,B 0,C 180,E1 -11484.872,E2 -11484.872} C_VEL
LIN {X 0,Y 391.422,Z 254.309,A -85,B 0,C 180,E1 -11485.955,E2 -11485.955} C_VEL
LIN {X 0,Y 392.04,Z 244.724,A -85,B 0,C 180,E1 -11486.975,E2 -11486.975} C_VEL
LIN {X 0,Y 392.599,Z 235.589,A -85,B 0,C 180,E1 -11487.718,E2 -11487.718} C_VEL
LIN {X 0,Y 391.635,Z 228.88,A -85,B 0,C 180,E1 -11488.211,E2 -11488.211} C_VEL
LIN {X 0,Y 389.86,Z 220.052,A -85,B 0,C 180,E1 -11488.747,E2 -11488.747} C_VEL
LIN {X 0,Y 389.098,Z 216.481,A -85,B 0,C 180,E1 -11488.944,E2 -11488.944} C_VEL
LIN {X 0,Y 389.231,Z 212.071,A -85,B 0,C 180,E1 -11492.221,E2 -11492.221} C_VEL
LIN {X 0,Y 389.371,Z 207.799,A -85,B 0,C 180,E1 -11495.473,E2 -11495.473} C_VEL
LIN {X 0,Y 389.613,Z 203.418,A -85,B 0,C 180,E1 -11498.854,E2 -11498.854} C_VEL
LIN {X 0,Y 389.82,Z 199.254,A -85,B 0,C 180,E1 -11502.153,E2 -11502.153} C_VEL
LIN {X 0,Y 390.046,Z 195.27,A -85,B 0,C 180,E1 -11505.39,E2 -11505.39} C_VEL
LIN {X 0,Y 390.104,Z 192.765,A -85,B 0,C 180,E1 -11507.516,E2 -11507.516} C_VEL
LIN {X 0,Y 390.204,Z 192.695,A -85,B 0,C 180,E1 -11510.672,E2 -11510.672} C_VEL
LIN {X 0,Y 390.319,Z 192.685,A -85,B 0,C 180,E1 -11512.76,E2 -11512.76} C_VEL
LIN {X 0,Y 390.227,Z 192.696,A -85,B 0,C 180,E1 -11514.834,E2 -11514.834} C_VEL
LIN {X 0,Y 390.419,Z 192.669,A -85,B 0,C 180,E1 -11517.938,E2 -11517.938} C_VEL
LIN {X 0,Y 390.552,Z 192.651,A -85,B 0,C 180,E1 -11520.001,E2 -11520.001} C_VEL
LIN {X 0,Y 390.311,Z 192.678,A -85,B 0,C 180,E1 -11523.097,E2 -11523.097} C_VEL
LIN {X 0,Y 390.323,Z 192.679,A -85,B 0,C 180,E1 -11526.203,E2 -11526.203} C_VEL
LIN {X 0,Y 390.195,Z 192.695,A -85,B 0,C 180,E1 -11529.33,E2 -11529.33} C_VEL
LIN {X 0,Y 390.173,Z 192.698,A -85,B 0,C 180,E1 -11532.484,E2 -11532.484} C_VEL
LIN {X 0,Y 390.142,Z 192.701,A -85,B 0,C 180,E1 -11535.677,E2 -11535.677} C_VEL
LIN {X 0,Y 390.108,Z 192.705,A -85,B 0,C 180,E1 -11538.923,E2 -11538.923} C_VEL
LIN {X 0,Y 390.042,Z 192.714,A -85,B 0,C 180,E1 -11542.235,E2 -11542.235} C_VEL
LIN {X 0,Y 390.121,Z 192.701,A -85,B 0,C 180,E1 -11545.744,E2 -11545.744} C_VEL
LIN {X 0,Y 390.061,Z 192.712,A -85,B 0,C 180,E1 -11549.11,E2 -11549.11} C_VEL
LIN {X 0,Y 390.045,Z 192.712,A -85,B 0,C 180,E1 -11552.722,E2 -11552.722} C_VEL
LIN {X 0,Y 390.058,Z 192.712,A -85,B 0,C 180,E1 -11555.826,E2 -11555.826} C_VEL
LIN {X 0,Y 390.071,Z 192.712,A -85,B 0,C 180,E1 -11559.218,E2 -11559.218} C_VEL
LIN {X 0,Y 390.045,Z 192.717,A -85,B 0,C 180,E1 -11562.375,E2 -11562.375} C_VEL
LIN {X 0,Y 390.046,Z 192.716,A -85,B 0,C 180,E1 -11565.355,E2 -11565.355} C_VEL
LIN {X 0,Y 390.033,Z 192.718,A -85,B 0,C 180,E1 -11568.187,E2 -11568.187} C_VEL
LIN {X 0,Y 390.071,Z 192.719,A -85,B 0,C 180,E1 -11571.732,E2 -11571.732} C_VEL
LIN {X 0,Y 391.091,Z 198.069,A -85,B 0,C 180,E1 -11574.897,E2 -11574.897} C_VEL
LIN {X 0,Y 392.043,Z 203.929,A -85,B 0,C 180,E1 -11578.073,E2 -11578.073} C_VEL
LIN {X 0,Y 391.679,Z 208.734,A -85,B 0,C 180,E1 -11580.433,E2 -11580.433} C_VEL
LIN {X 0,Y 390.79,Z 216.538,A -85,B 0,C 180,E1 -11584.054,E2 -11584.054} C_VEL
LIN {X 0,Y 390.183,Z 223.661,A -85,B 0,C 180,E1 -11587.224,E2 -11587.224} C_VEL
LIN {X 0,Y 389.712,Z 231.271,A -85,B 0,C 180,E1 -11590.511,E2 -11590.511} C_VEL
LIN {X 0,Y 389.226,Z 240.305,A -85,B 0,C 180,E1 -11594.286,E2 -11594.286} C_VEL
LIN {X 0,Y 389.123,Z 242.562,A -85,B 0,C 180,E1 -11595.22,E2 -11595.22} C_VEL
LIN {X 0,Y 390.963,Z 256.042,A -85,B 0,C 180,E1 -11595.876,E2 -11595.876} C_VEL
LIN {X 0,Y 391.624,Z 264.596,A -85,B 0,C 180,E1 -11596.416,E2 -11596.416} C_VEL
LIN {X 0,Y 391.726,Z 272.754,A -85,B 0,C 180,E1 -11597.041,E2 -11597.041} C_VEL
LIN {X 0,Y 391.098,Z 281.099,A -85,B 0,C 180,E1 -11597.811,E2 -11597.811} C_VEL
LIN {X 0,Y 390.561,Z 289.012,A -85,B 0,C 180,E1 -11598.715,E2 -11598.715} C_VEL
LIN {X 0,Y 390.073,Z 295.566,A -85,B 0,C 180,E1 -11599.62,E2 -11599.62} C_VEL
LIN {X 0,Y 389.646,Z 301.81,A -85,B 0,C 180,E1 -11600.658,E2 -11600.658} C_VEL
LIN {X 0,Y 389.295,Z 306.998,A -85,B 0,C 180,E1 -11601.696,E2 -11601.696} C_VEL
LIN {X 0,Y 389.051,Z 311.321,A -85,B 0,C 180,E1 -11602.736,E2 -11602.736} C_VEL
LIN {X 0,Y 388.835,Z 314.908,A -85,B 0,C 180,E1 -11603.774,E2 -11603.774} C_VEL
LIN {X 0,Y 388.788,Z 319.036,A -85,B 0,C 180,E1 -11605.334,E2 -11605.334} C_VEL
LIN {X 0,Y 388.69,Z 321.888,A -85,B 0,C 180,E1 -11606.891,E2 -11606.891} C_VEL
LIN {X 0,Y 388.759,Z 323.058,A -85,B 0,C 180,E1 -11607.928,E2 -11607.928} C_VEL
LIN {X 0,Y 388.761,Z 323.74,A -85,B 0,C 180,E1 -11608.964,E2 -11608.964} C_VEL
LIN {X 0,Y 388.749,Z 323.944,A -85,B 0,C 180,E1 -11610,E2 -11610} C_VEL
LIN {X 0,Y 388.761,Z 323.633,A -85,B 0,C 180,E1 -11611.036,E2 -11611.036} C_VEL
LIN {X 0,Y 388.777,Z 322.725,A -85,B 0,C 180,E1 -11612.072,E2 -11612.072} C_VEL
LIN {X 0,Y 388.707,Z 321.301,A -85,B 0,C 180,E1 -11613.11,E2 -11613.11} C_VEL
LIN {X 0,Y 388.808,Z 318.207,A -85,B 0,C 180,E1 -11614.666,E2 -11614.666} C_VEL
LIN {X 0,Y 388.835,Z 313.711,A -85,B 0,C 180,E1 -11616.226,E2 -11616.226} C_VEL
LIN {X 0,Y 389.092,Z 308.696,A -85,B 0,C 180,E1 -11617.525,E2 -11617.525} C_VEL
LIN {X 0,Y 389.33,Z 303.793,A -85,B 0,C 180,E1 -11618.565,E2 -11618.565} C_VEL
LIN {X 0,Y 389.643,Z 297.866,A -85,B 0,C 180,E1 -11619.605,E2 -11619.605} C_VEL
LIN {X 0,Y 390.119,Z 290.648,A -85,B 0,C 180,E1 -11620.641,E2 -11620.641} C_VEL
LIN {X 0,Y 390.443,Z 284.157,A -85,B 0,C 180,E1 -11621.42,E2 -11621.42} C_VEL
LIN {X 0,Y 390.971,Z 276.323,A -85,B 0,C 180,E1 -11622.194,E2 -11622.194} C_VEL
LIN {X 0,Y 391.263,Z 269.093,A -85,B 0,C 180,E1 -11622.784,E2 -11622.784} C_VEL
LIN {X 0,Y 390.761,Z 260.511,A -85,B 0,C 180,E1 -11623.364,E2 -11623.364} C_VEL
LIN {X 0,Y 389.823,Z 250.845,A -85,B 0,C 180,E1 -11623.869,E2 -11623.869} C_VEL
LIN {X 0,Y 389.03,Z 243.393,A -85,B 0,C 180,E1 -11624.173,E2 -11624.173} C_VEL
LIN {X 0,Y 389.36,Z 235.876,A -85,B 0,C 180,E1 -11627.273,E2 -11627.273} C_VEL
LIN {X 0,Y 389.732,Z 228.553,A -85,B 0,C 180,E1 -11630.329,E2 -11630.329} C_VEL
LIN {X 0,Y 390.294,Z 220.146,A -85,B 0,C 180,E1 -11633.901,E2 -11633.901} C_VEL
LIN {X 0,Y 390.959,Z 212.334,A -85,B 0,C 180,E1 -11637.284,E2 -11637.284} C_VEL
LIN {X 0,Y 391.657,Z 205.031,A -85,B 0,C 180,E1 -11640.534,E2 -11640.534} C_VEL
LIN {X 0,Y 391.709,Z 202.056,A -85,B 0,C 180,E1 -11641.904,E2 -11641.904} C_VEL
LIN {X 0,Y 390.595,Z 195.38,A -85,B 0,C 180,E1 -11645.154,E2 -11645.154} C_VEL
LIN {X 0,Y 390.08,Z 192.71,A -85,B 0,C 180,E1 -11646.562,E2 -11646.562} C_VEL
LIN {X 0,Y 390.072,Z 192.715,A -85,B 0,C 180,E1 -11649.218,E2 -11649.218} C_VEL
LIN {X 0,Y 390.046,Z 192.714,A -85,B 0,C 180,E1 -11652.374,E2 -11652.374} C_VEL
LIN {X 0,Y 390.048,Z 192.71,A -85,B 0,C 180,E1 -11655.354,E2 -11655.354} C_VEL
LIN {X 0,Y 390.028,Z 192.717,A -85,B 0,C 180,E1 -11658.186,E2 -11658.186} C_VEL
LIN {X 0,Y 390.067,Z 192.708,A -85,B 0,C 180,E1 -11660.904,E2 -11660.904} C_VEL
LIN {X 0,Y 390.089,Z 192.705,A -85,B 0,C 180,E1 -11664.793,E2 -11664.793} C_VEL
LIN {X 0,Y 390.028,Z 192.714,A -85,B 0,C 180,E1 -11668.495,E2 -11668.495} C_VEL
LIN {X 0,Y 390.122,Z 192.705,A -85,B 0,C 180,E1 -11672.07,E2 -11672.07} C_VEL
LIN {X 0,Y 390.082,Z 192.708,A -85,B 0,C 180,E1 -11675.519,E2 -11675.519} C_VEL
LIN {X 0,Y 390.092,Z 192.708,A -85,B 0,C 180,E1 -11679.529,E2 -11679.529} C_VEL
LIN {X 0,Y 390.143,Z 192.7,A -85,B 0,C 180,E1 -11683.248,E2 -11683.248} C_VEL
LIN {X 0,Y 390.199,Z 192.691,A -85,B 0,C 180,E1 -11686.561,E2 -11686.561} C_VEL
LIN {X 0,Y 390.171,Z 192.699,A -85,B 0,C 180,E1 -11689.622,E2 -11689.622} C_VEL
LIN {X 0,Y 390.285,Z 192.682,A -85,B 0,C 180,E1 -11692.758,E2 -11692.758} C_VEL
LIN {X 0,Y 390.226,Z 192.689,A -85,B 0,C 180,E1 -11694.833,E2 -11694.833} C_VEL
LIN {X 0,Y 390.421,Z 192.664,A -85,B 0,C 180,E1 -11697.936,E2 -11697.936} C_VEL
LIN {X 0,Y 390.55,Z 192.648,A -85,B 0,C 180,E1 -11699.999,E2 -11699.999} C_VEL
LIN {X 0,Y 390.313,Z 192.681,A -85,B 0,C 180,E1 -11703.096,E2 -11703.096} C_VEL
LIN {X 0,Y 390.289,Z 192.679,A -85,B 0,C 180,E1 -11706.64,E2 -11706.64} C_VEL
LIN {X 0,Y 390.195,Z 192.693,A -85,B 0,C 180,E1 -11709.328,E2 -11709.328} C_VEL
LIN {X 0,Y 390.173,Z 192.697,A -85,B 0,C 180,E1 -11712.482,E2 -11712.482} C_VEL
LIN {X 0,Y 390.14,Z 192.699,A -85,B 0,C 180,E1 -11715.676,E2 -11715.676} C_VEL
LIN {X 0,Y 390.103,Z 192.707,A -85,B 0,C 180,E1 -11718.921,E2 -11718.921} C_VEL
LIN {X 0,Y 390.038,Z 192.714,A -85,B 0,C 180,E1 -11722.233,E2 -11722.233} C_VEL
LIN {X 0,Y 390.118,Z 192.702,A -85,B 0,C 180,E1 -11725.742,E2 -11725.742} C_VEL
LIN {X 0,Y 390.057,Z 192.71,A -85,B 0,C 180,E1 -11729.108,E2 -11729.108} C_VEL
LIN {X 0,Y 390.041,Z 192.713,A -85,B 0,C 180,E1 -11732.72,E2 -11732.72} C_VEL
LIN {X 0,Y 390.055,Z 192.711,A -85,B 0,C 180,E1 -11735.824,E2 -11735.824} C_VEL
LIN {X 0,Y 390.067,Z 192.707,A -85,B 0,C 180,E1 -11739.217,E2 -11739.217} C_VEL
LIN {X 0,Y 390.039,Z 192.713,A -85,B 0,C 180,E1 -11742.373,E2 -11742.373} C_VEL
LIN {X 0,Y 390.039,Z 192.712,A -85,B 0,C 180,E1 -11745.353,E2 -11745.353} C_VEL
LIN {X 0,Y 390.026,Z 192.716,A -85,B 0,C 180,E1 -11748.186,E2 -11748.186} C_VEL
LIN {X 0,Y 390.085,Z 192.705,A -85,B 0,C 180,E1 -11750.907,E2 -11750.907} C_VEL
LIN {X 0,Y 390.08,Z 192.706,A -85,B 0,C 180,E1 -11754.792,E2 -11754.792} C_VEL
LIN {X 0,Y 390.028,Z 192.715,A -85,B 0,C 180,E1 -11757.874,E2 -11757.874} C_VEL
LIN {X 0,Y 390.059,Z 192.709,A -85,B 0,C 180,E1 -11760.89,E2 -11760.89} C_VEL
LIN {X 0,Y 390.104,Z 192.703,A -85,B 0,C 180,E1 -11764.381,E2 -11764.381} C_VEL
LIN {X 0,Y 390.033,Z 192.714,A -85,B 0,C 180,E1 -11767.765,E2 -11767.765} C_VEL
LIN {X 0,Y 390.098,Z 192.707,A -85,B 0,C 180,E1 -11771.077,E2 -11771.077} C_VEL
LIN {X 0,Y 390.132,Z 192.7,A -85,B 0,C 180,E1 -11774.323,E2 -11774.323} C_VEL
LIN {X 0,Y 390.171,Z 192.697,A -85,B 0,C 180,E1 -11777.517,E2 -11777.517} C_VEL
LIN {X 0,Y 390.306,Z 192.678,A -85,B 0,C 180,E1 -11781.717,E2 -11781.717} C_VEL
LIN {X 0,Y 390.321,Z 192.675,A -85,B 0,C 180,E1 -11783.798,E2 -11783.798} C_VEL
LIN {X 0,Y 390.409,Z 192.665,A -85,B 0,C 180,E1 -11787.937,E2 -11787.937} C_VEL
LIN {X 0,Y 390.541,Z 192.649,A -85,B 0,C 180,E1 -11790,E2 -11790} C_VEL
LIN {X 0,Y 390.307,Z 192.68,A -85,B 0,C 180,E1 -11793.096,E2 -11793.096} C_VEL
LIN {X 0,Y 390.321,Z 192.679,A -85,B 0,C 180,E1 -11796.202,E2 -11796.202} C_VEL
LIN {X 0,Y 390.305,Z 192.681,A -85,B 0,C 180,E1 -11798.282,E2 -11798.282} C_VEL
LIN {X 0,Y 390.117,Z 192.701,A -85,B 0,C 180,E1 -11801.43,E2 -11801.43} C_VEL
LIN {X 0,Y 389.886,Z 192.735,A -85,B 0,C 180,E1 -11804.617,E2 -11804.617} C_VEL
LIN {X 0,Y 389.737,Z 193.017,A -85,B 0,C 180,E1 -11805.425,E2 -11805.425} C_VEL
LIN {X 0,Y 389.468,Z 197.702,A -85,B 0,C 180,E1 -11808.954,E2 -11808.954} C_VEL
LIN {X 0,Y 389.324,Z 202.204,A -85,B 0,C 180,E1 -11812.277,E2 -11812.277} C_VEL
LIN {X 0,Y 389.167,Z 206.914,A -85,B 0,C 180,E1 -11815.685,E2 -11815.685} C_VEL
LIN {X 0,Y 388.97,Z 211.863,A -85,B 0,C 180,E1 -11819.199,E2 -11819.199} C_VEL
LIN {X 0,Y 388.914,Z 213.611,A -85,B 0,C 180,E1 -11820.437,E2 -11820.437} C_VEL
LIN {X 0,Y 388.717,Z 215.067,A -85,B 0,C 180,E1 -11820.947,E2 -11820.947} C_VEL
LIN {X 0,Y 388.273,Z 217.486,A -85,B 0,C 180,E1 -11821.375,E2 -11821.375} C_VEL
LIN {X 0,Y 387.342,Z 222.186,A -85,B 0,C 180,E1 -11821.881,E2 -11821.881} C_VEL
LIN {X 0,Y 384.986,Z 235.584,A -85,B 0,C 180,E1 -11822.761,E2 -11822.761} C_VEL
LIN {X 0,Y 384.613,Z 239.37,A -85,B 0,C 180,E1 -11823.053,E2 -11823.053} C_VEL
LIN {X 0,Y 384.107,Z 248.631,A -85,B 0,C 180,E1 -11823.921,E2 -11823.921} C_VEL
LIN {X 0,Y 383.69,Z 255.82,A -85,B 0,C 180,E1 -11824.758,E2 -11824.758} C_VEL
LIN {X 0,Y 383.19,Z 262.984,A -85,B 0,C 180,E1 -11825.776,E2 -11825.776} C_VEL
LIN {X 0,Y 382.748,Z 269.956,A -85,B 0,C 180,E1 -11827.001,E2 -11827.001} C_VEL
LIN {X 0,Y 382.411,Z 275.401,A -85,B 0,C 180,E1 -11828.215,E2 -11828.215} C_VEL
LIN {X 0,Y 382.079,Z 279.689,A -85,B 0,C 180,E1 -11829.419,E2 -11829.419} C_VEL
LIN {X 0,Y 381.796,Z 283.893,A -85,B 0,C 180,E1 -11831.001,E2 -11831.001} C_VEL
LIN {X 0,Y 381.66,Z 286.736,A -85,B 0,C 180,E1 -11832.562,E2 -11832.562} C_VEL
LIN {X 0,Y 381.527,Z 288.449,A -85,B 0,C 180,E1 -11834.426,E2 -11834.426} C_VEL
LIN {X 0,Y 381.527,Z 288.599,A -85,B 0,C 180,E1 -11835.923,E2 -11835.923} C_VEL
LIN {X 0,Y 381.676,Z 287.671,A -85,B 0,C 180,E1 -11837.437,E2 -11837.437} C_VEL
LIN {X 0,Y 381.912,Z 285.599,A -85,B 0,C 180,E1 -11838.981,E2 -11838.981} C_VEL
LIN {X 0,Y 382.219,Z 282.085,A -85,B 0,C 180,E1 -11840.558,E2 -11840.558} C_VEL
LIN {X 0,Y 382.566,Z 278.343,A -85,B 0,C 180,E1 -11841.787,E2 -11841.787} C_VEL
LIN {X 0,Y 382.942,Z 273.623,A -85,B 0,C 180,E1 -11843.006,E2 -11843.006} C_VEL
LIN {X 0,Y 383.367,Z 268.464,A -85,B 0,C 180,E1 -11844.083,E2 -11844.083} C_VEL
LIN {X 0,Y 383.892,Z 262.492,A -85,B 0,C 180,E1 -11845.105,E2 -11845.105} C_VEL
LIN {X 0,Y 384.48,Z 255.277,A -85,B 0,C 180,E1 -11846.117,E2 -11846.117} C_VEL
LIN {X 0,Y 385.148,Z 245.51,A -85,B 0,C 180,E1 -11847.199,E2 -11847.199} C_VEL
LIN {X 0,Y 385.741,Z 236.509,A -85,B 0,C 180,E1 -11847.953,E2 -11847.953} C_VEL
LIN {X 0,Y 384.378,Z 227.91,A -85,B 0,C 180,E1 -11848.596,E2 -11848.596} C_VEL
LIN {X 0,Y 382.389,Z 218.603,A -85,B 0,C 180,E1 -11849.158,E2 -11849.158} C_VEL
LIN {X 0,Y 382.007,Z 216.748,A -85,B 0,C 180,E1 -11849.285,E2 -11849.285} C_VEL
LIN {X 0,Y 382.176,Z 212.337,A -85,B 0,C 180,E1 -11852.631,E2 -11852.631} C_VEL
LIN {X 0,Y 382.358,Z 207.775,A -85,B 0,C 180,E1 -11856.149,E2 -11856.149} C_VEL
LIN {X 0,Y 382.611,Z 203.471,A -85,B 0,C 180,E1 -11859.575,E2 -11859.575} C_VEL
LIN {X 0,Y 382.893,Z 199.319,A -85,B 0,C 180,E1 -11862.923,E2 -11862.923} C_VEL
LIN {X 0,Y 383.112,Z 195.084,A -85,B 0,C 180,E1 -11866.473,E2 -11866.473} C_VEL
LIN {X 0,Y 383.107,Z 194.149,A -85,B 0,C 180,E1 -11867.284,E2 -11867.284} C_VEL
LIN {X 0,Y 383.06,Z 193.589,A -85,B 0,C 180,E1 -11868.358,E2 -11868.358} C_VEL
LIN {X 0,Y 383.307,Z 193.557,A -85,B 0,C 180,E1 -11871.931,E2 -11871.931} C_VEL
LIN {X 0,Y 383.2,Z 193.572,A -85,B 0,C 180,E1 -11874.739,E2 -11874.739} C_VEL
LIN {X 0,Y 383.387,Z 193.544,A -85,B 0,C 180,E1 -11877.9,E2 -11877.9} C_VEL
LIN {X 0,Y 383.521,Z 193.526,A -85,B 0,C 180,E1 -11880.001,E2 -11880.001} C_VEL
LIN {X 0,Y 383.248,Z 193.558,A -85,B 0,C 180,E1 -11883.155,E2 -11883.155} C_VEL
LIN {X 0,Y 383.278,Z 193.556,A -85,B 0,C 180,E1 -11886.317,E2 -11886.317} C_VEL
LIN {X 0,Y 383.145,Z 193.574,A -85,B 0,C 180,E1 -11889.503,E2 -11889.503} C_VEL
LIN {X 0,Y 383.138,Z 193.575,A -85,B 0,C 180,E1 -11892.717,E2 -11892.717} C_VEL
LIN {X 0,Y 383.083,Z 193.581,A -85,B 0,C 180,E1 -11895.974,E2 -11895.974} C_VEL
LIN {X 0,Y 383.063,Z 193.582,A -85,B 0,C 180,E1 -11899.284,E2 -11899.284} C_VEL
LIN {X 0,Y 383.04,Z 193.586,A -85,B 0,C 180,E1 -11903.451,E2 -11903.451} C_VEL
LIN {X 0,Y 383.082,Z 193.579,A -85,B 0,C 180,E1 -11906.124,E2 -11906.124} C_VEL
LIN {X 0,Y 382.994,Z 193.592,A -85,B 0,C 180,E1 -11909.7,E2 -11909.7} C_VEL
LIN {X 0,Y 383.005,Z 193.591,A -85,B 0,C 180,E1 -11913.401,E2 -11913.401} C_VEL
LIN {X 0,Y 383.034,Z 193.586,A -85,B 0,C 180,E1 -11916.165,E2 -11916.165} C_VEL
LIN {X 0,Y 383.01,Z 193.591,A -85,B 0,C 180,E1 -11919.959,E2 -11919.959} C_VEL
LIN {X 0,Y 383.007,Z 193.593,A -85,B 0,C 180,E1 -11922.779,E2 -11922.779} C_VEL
LIN {X 0,Y 382.999,Z 193.595,A -85,B 0,C 180,E1 -11925.79,E2 -11925.79} C_VEL
LIN {X 0,Y 382.99,Z 193.594,A -85,B 0,C 180,E1 -11928.796,E2 -11928.796} C_VEL
LIN {X 0,Y 383.061,Z 193.738,A -85,B 0,C 180,E1 -11931.406,E2 -11931.406} C_VEL
LIN {X 0,Y 384.106,Z 199.33,A -85,B 0,C 180,E1 -11934.806,E2 -11934.806} C_VEL
LIN {X 0,Y 384.836,Z 203.495,A -85,B 0,C 180,E1 -11937.148,E2 -11937.148} C_VEL
LIN {X 0,Y 385.071,Z 206.333,A -85,B 0,C 180,E1 -11938.634,E2 -11938.634} C_VEL
LIN {X 0,Y 384.363,Z 212.384,A -85,B 0,C 180,E1 -11941.614,E2 -11941.614} C_VEL
LIN {X 0,Y 383.553,Z 219.806,A -85,B 0,C 180,E1 -11945.075,E2 -11945.075} C_VEL
LIN {X 0,Y 382.922,Z 227.344,A -85,B 0,C 180,E1 -11948.465,E2 -11948.465} C_VEL
LIN {X 0,Y 382.417,Z 234.971,A -85,B 0,C 180,E1 -11951.795,E2 -11951.795} C_VEL
LIN {X 0,Y 382.059,Z 242.297,A -85,B 0,C 180,E1 -11954.906,E2 -11954.906} C_VEL
LIN {X 0,Y 383.944,Z 255.63,A -85,B 0,C 180,E1 -11955.565,E2 -11955.565} C_VEL
LIN {X 0,Y 384.692,Z 264.198,A -85,B 0,C 180,E1 -11956.122,E2 -11956.122} C_VEL
LIN {X 0,Y 384.864,Z 271.35,A -85,B 0,C 180,E1 -11956.671,E2 -11956.671} C_VEL
LIN {X 0,Y 384.305,Z 279.867,A -85,B 0,C 180,E1 -11957.458,E2 -11957.458} C_VEL
LIN {X 0,Y 383.65,Z 287.915,A -85,B 0,C 180,E1 -11958.375,E2 -11958.375} C_VEL
LIN {X 0,Y 383.232,Z 293.726,A -85,B 0,C 180,E1 -11959.166,E2 -11959.166} C_VEL
LIN {X 0,Y 382.707,Z 300.214,A -85,B 0,C 180,E1 -11960.22,E2 -11960.22} C_VEL
LIN {X 0,Y 382.348,Z 305.621,A -85,B 0,C 180,E1 -11961.278,E2 -11961.278} C_VEL
LIN {X 0,Y 381.989,Z 311.108,A -85,B 0,C 180,E1 -11962.601,E2 -11962.601} C_VEL
LIN {X 0,Y 381.738,Z 315.122,A -85,B 0,C 180,E1 -11963.812,E2 -11963.812} C_VEL
LIN {X 0,Y 381.698,Z 318.78,A -85,B 0,C 180,E1 -11965.247,E2 -11965.247} C_VEL
LIN {X 0,Y 381.598,Z 321.612,A -85,B 0,C 180,E1 -11966.833,E2 -11966.833} C_VEL
LIN {X 0,Y 381.657,Z 322.761,A -85,B 0,C 180,E1 -11967.89,E2 -11967.89} C_VEL
LIN {X 0,Y 381.692,Z 323.422,A -85,B 0,C 180,E1 -11968.945,E2 -11968.945} C_VEL
LIN {X 0,Y 381.678,Z 323.605,A -85,B 0,C 180,E1 -11970,E2 -11970} C_VEL
LIN {X 0,Y 381.692,Z 323.284,A -85,B 0,C 180,E1 -11971.055,E2 -11971.055} C_VEL
LIN {X 0,Y 381.677,Z 322.363,A -85,B 0,C 180,E1 -11972.111,E2 -11972.111} C_VEL
LIN {X 0,Y 381.614,Z 320.913,A -85,B 0,C 180,E1 -11973.167,E2 -11973.167} C_VEL
LIN {X 0,Y 381.717,Z 317.793,A -85,B 0,C 180,E1 -11974.753,E2 -11974.753} C_VEL
LIN {X 0,Y 381.771,Z 313.237,A -85,B 0,C 180,E1 -11976.342,E2 -11976.342} C_VEL
LIN {X 0,Y 382.031,Z 308.184,A -85,B 0,C 180,E1 -11977.665,E2 -11977.665} C_VEL
LIN {X 0,Y 382.278,Z 303.239,A -85,B 0,C 180,E1 -11978.724,E2 -11978.724} C_VEL
LIN {X 0,Y 382.621,Z 297.265,A -85,B 0,C 180,E1 -11979.782,E2 -11979.782} C_VEL
LIN {X 0,Y 383.134,Z 289.99,A -85,B 0,C 180,E1 -11980.838,E2 -11980.838} C_VEL
LIN {X 0,Y 383.483,Z 283.428,A -85,B 0,C 180,E1 -11981.63,E2 -11981.63} C_VEL
LIN {X 0,Y 384.014,Z 275.5,A -85,B 0,C 180,E1 -11982.418,E2 -11982.418} C_VEL
LIN {X 0,Y 384.242,Z 268.551,A -85,B 0,C 180,E1 -11982.992,E2 -11982.992} C_VEL
LIN {X 0,Y 383.647,Z 259.164,A -85,B 0,C 180,E1 -11983.627,E2 -11983.627} C_VEL
LIN {X 0,Y 382.623,Z 249.332,A -85,B 0,C 180,E1 -11984.137,E2 -11984.137} C_VEL
LIN {X 0,Y 381.973,Z 243.169,A -85,B 0,C 180,E1 -11984.382,E2 -11984.382} C_VEL
LIN {X 0,Y 382.318,Z 235.41,A -85,B 0,C 180,E1 -11987.657,E2 -11987.657} C_VEL
LIN {X 0,Y 382.743,Z 227.627,A -85,B 0,C 180,E1 -11990.981,E2 -11990.981} C_VEL
LIN {X 0,Y 383.3,Z 219.828,A -85,B 0,C 180,E1 -11994.365,E2 -11994.365} C_VEL
LIN {X 0,Y 384.033,Z 212.061,A -85,B 0,C 180,E1 -11997.818,E2 -11997.818} C_VEL
LIN {X 0,Y 384.771,Z 204.279,A -85,B 0,C 180,E1 -12001.37,E2 -12001.37} C_VEL
LIN {X 0,Y 384.062,Z 199.116,A -85,B 0,C 180,E1 -12003.893,E2 -12003.893} C_VEL
LIN {X 0,Y 383.041,Z 193.587,A -85,B 0,C 180,E1 -12006.83,E2 -12006.83} C_VEL
LIN {X 0,Y 383.012,Z 193.588,A -85,B 0,C 180,E1 -12009.958,E2 -12009.958} C_VEL
LIN {X 0,Y 383.009,Z 193.589,A -85,B 0,C 180,E1 -12012.778,E2 -12012.778} C_VEL
LIN {X 0,Y 383,Z 193.589,A -85,B 0,C 180,E1 -12015.789,E2 -12015.789} C_VEL
LIN {X 0,Y 382.974,Z 193.593,A -85,B 0,C 180,E1 -12018.799,E2 -12018.799} C_VEL
LIN {X 0,Y 382.999,Z 193.592,A -85,B 0,C 180,E1 -12022.097,E2 -12022.097} C_VEL
LIN {X 0,Y 383.022,Z 193.585,A -85,B 0,C 180,E1 -12025.332,E2 -12025.332} C_VEL
LIN {X 0,Y 382.987,Z 193.589,A -85,B 0,C 180,E1 -12029.081,E2 -12029.081} C_VEL
LIN {X 0,Y 383.061,Z 193.58,A -85,B 0,C 180,E1 -12032.698,E2 -12032.698} C_VEL
LIN {X 0,Y 383.055,Z 193.581,A -85,B 0,C 180,E1 -12035.039,E2 -12035.039} C_VEL
LIN {X 0,Y 382.997,Z 193.589,A -85,B 0,C 180,E1 -12038.469,E2 -12038.469} C_VEL
LIN {X 0,Y 383.093,Z 193.58,A -85,B 0,C 180,E1 -12041.827,E2 -12041.827} C_VEL
LIN {X 0,Y 383.115,Z 193.575,A -85,B 0,C 180,E1 -12045.118,E2 -12045.118} C_VEL
LIN {X 0,Y 383.101,Z 193.575,A -85,B 0,C 180,E1 -12048.357,E2 -12048.357} C_VEL
LIN {X 0,Y 383.232,Z 193.56,A -85,B 0,C 180,E1 -12052.013,E2 -12052.013} C_VEL
LIN {X 0,Y 383.198,Z 193.564,A -85,B 0,C 180,E1 -12054.738,E2 -12054.738} C_VEL
LIN {X 0,Y 383.388,Z 193.54,A -85,B 0,C 180,E1 -12057.898,E2 -12057.898} C_VEL
LIN {X 0,Y 383.519,Z 193.524,A -85,B 0,C 180,E1 -12059.999,E2 -12059.999} C_VEL
LIN {X 0,Y 383.249,Z 193.561,A -85,B 0,C 180,E1 -12063.153,E2 -12063.153} C_VEL
LIN {X 0,Y 383.248,Z 193.556,A -85,B 0,C 180,E1 -12066.63,E2 -12066.63} C_VEL
LIN {X 0,Y 383.145,Z 193.57,A -85,B 0,C 180,E1 -12069.501,E2 -12069.501} C_VEL
LIN {X 0,Y 383.127,Z 193.572,A -85,B 0,C 180,E1 -12073.535,E2 -12073.535} C_VEL
LIN {X 0,Y 383.095,Z 193.578,A -85,B 0,C 180,E1 -12077.068,E2 -12077.068} C_VEL
LIN {X 0,Y 383.029,Z 193.589,A -85,B 0,C 180,E1 -12080.646,E2 -12080.646} C_VEL
LIN {X 0,Y 383.022,Z 193.585,A -85,B 0,C 180,E1 -12083.807,E2 -12083.807} C_VEL
LIN {X 0,Y 383.079,Z 193.581,A -85,B 0,C 180,E1 -12086.122,E2 -12086.122} C_VEL
LIN {X 0,Y 383.039,Z 193.587,A -85,B 0,C 180,E1 -12088.491,E2 -12088.491} C_VEL
LIN {X 0,Y 383.008,Z 193.591,A -85,B 0,C 180,E1 -12092.148,E2 -12092.148} C_VEL
LIN {X 0,Y 383.016,Z 193.588,A -85,B 0,C 180,E1 -12094.667,E2 -12094.667} C_VEL
LIN {X 0,Y 382.998,Z 193.591,A -85,B 0,C 180,E1 -12097.903,E2 -12097.903} C_VEL
LIN {X 0,Y 382.98,Z 193.591,A -85,B 0,C 180,E1 -12101.346,E2 -12101.346} C_VEL
LIN {X 0,Y 382.991,Z 193.592,A -85,B 0,C 180,E1 -12104.302,E2 -12104.302} C_VEL
LIN {X 0,Y 383.005,Z 193.587,A -85,B 0,C 180,E1 -12107.239,E2 -12107.239} C_VEL
LIN {X 0,Y 383.01,Z 193.587,A -85,B 0,C 180,E1 -12110.412,E2 -12110.412} C_VEL
LIN {X 0,Y 383.021,Z 193.588,A -85,B 0,C 180,E1 -12114.044,E2 -12114.044} C_VEL
LIN {X 0,Y 382.982,Z 193.594,A -85,B 0,C 180,E1 -12117.577,E2 -12117.577} C_VEL
LIN {X 0,Y 382.991,Z 193.589,A -85,B 0,C 180,E1 -12120.3,E2 -12120.3} C_VEL
LIN {X 0,Y 383.05,Z 193.582,A -85,B 0,C 180,E1 -12122.697,E2 -12122.697} C_VEL
LIN {X 0,Y 383.026,Z 193.585,A -85,B 0,C 180,E1 -12126.192,E2 -12126.192} C_VEL
LIN {X 0,Y 383.047,Z 193.585,A -85,B 0,C 180,E1 -12129.598,E2 -12129.598} C_VEL
LIN {X 0,Y 383.097,Z 193.578,A -85,B 0,C 180,E1 -12132.931,E2 -12132.931} C_VEL
LIN {X 0,Y 383.117,Z 193.573,A -85,B 0,C 180,E1 -12136.463,E2 -12136.463} C_VEL
LIN {X 0,Y 383.133,Z 193.573,A -85,B 0,C 180,E1 -12139.43,E2 -12139.43} C_VEL
LIN {X 0,Y 383.265,Z 193.558,A -85,B 0,C 180,E1 -12142.625,E2 -12142.625} C_VEL
LIN {X 0,Y 383.19,Z 193.568,A -85,B 0,C 180,E1 -12144.738,E2 -12144.738} C_VEL
LIN {X 0,Y 383.376,Z 193.541,A -85,B 0,C 180,E1 -12147.899,E2 -12147.899} C_VEL
LIN {X 0,Y 383.51,Z 193.525,A -85,B 0,C 180,E1 -12150,E2 -12150} C_VEL
LIN {X 0,Y 383.243,Z 193.559,A -85,B 0,C 180,E1 -12153.154,E2 -12153.154} C_VEL
LIN {X 0,Y 383.278,Z 193.557,A -85,B 0,C 180,E1 -12156.316,E2 -12156.316} C_VEL
LIN {X 0,Y 383.251,Z 193.561,A -85,B 0,C 180,E1 -12158.436,E2 -12158.436} C_VEL
LIN {X 0,Y 383.057,Z 193.581,A -85,B 0,C 180,E1 -12161.643,E2 -12161.643} C_VEL
LIN {X 0,Y 382.943,Z 193.596,A -85,B 0,C 180,E1 -12163.803,E2 -12163.803} C_VEL
LIN {X 0,Y 382.723,Z 193.691,A -85,B 0,C 180,E1 -12165.306,E2 -12165.306} C_VEL
LIN {X 0,Y 382.465,Z 197.488,A -85,B 0,C 180,E1 -12168.203,E2 -12168.203} C_VEL
LIN {X 0,Y 382.281,Z 201.972,A -85,B 0,C 180,E1 -12171.573,E2 -12171.573} C_VEL
LIN {X 0,Y 382.132,Z 206.681,A -85,B 0,C 180,E1 -12175.024,E2 -12175.024} C_VEL
LIN {X 0,Y 381.928,Z 211.588,A -85,B 0,C 180,E1 -12178.583,E2 -12178.583} C_VEL
LIN {X 0,Y 381.869,Z 215.81,A -85,B 0,C 180,E1 -12181.578,E2 -12181.578} C_VEL
LIN {X 0,Y 383.514,Z 225.841,A -85,B 0,C 180,E1 -12182.102,E2 -12182.102} C_VEL
LIN {X 0,Y 384.658,Z 233.677,A -85,B 0,C 180,E1 -12182.627,E2 -12182.627} C_VEL
LIN {X 0,Y 384.613,Z 239.37,A -85,B 0,C 180,E1 -12183.053,E2 -12183.053} C_VEL
LIN {X 0,Y 383.649,Z 244.631,A -85,B 0,C 180,E1 -12183.496,E2 -12183.496} C_VEL
LIN {X 0,Y 380.324,Z 252.627,A -85,B 0,C 180,E1 -12184.252,E2 -12184.252} C_VEL
LIN {X 0,Y 377.052,Z 259.823,A -85,B 0,C 180,E1 -12185.114,E2 -12185.114} C_VEL
LIN {X 0,Y 376.109,Z 263.882,A -85,B 0,C 180,E1 -12185.731,E2 -12185.731} C_VEL
LIN {X 0,Y 375.638,Z 271.316,A -85,B 0,C 180,E1 -12187.109,E2 -12187.109} C_VEL
LIN {X 0,Y 375.245,Z 277.135,A -85,B 0,C 180,E1 -12188.517,E2 -12188.517} C_VEL
LIN {X 0,Y 374.908,Z 281.227,A -85,B 0,C 180,E1 -12189.775,E2 -12189.775} C_VEL
LIN {X 0,Y 374.708,Z 284.358,A -85,B 0,C 180,E1 -12191.03,E2 -12191.03} C_VEL
LIN {X 0,Y 374.526,Z 287.596,A -85,B 0,C 180,E1 -12192.961,E2 -12192.961} C_VEL
LIN {X 0,Y 374.43,Z 288.794,A -85,B 0,C 180,E1 -12194.502,E2 -12194.502} C_VEL
LIN {X 0,Y 374.44,Z 288.922,A -85,B 0,C 180,E1 -12196.017,E2 -12196.017} C_VEL
LIN {X 0,Y 374.596,Z 288.015,A -85,B 0,C 180,E1 -12197.515,E2 -12197.515} C_VEL
LIN {X 0,Y 374.826,Z 286.107,A -85,B 0,C 180,E1 -12198.987,E2 -12198.987} C_VEL
LIN {X 0,Y 375.126,Z 283.16,A -85,B 0,C 180,E1 -12200.434,E2 -12200.434} C_VEL
LIN {X 0,Y 375.524,Z 279.029,A -85,B 0,C 180,E1 -12201.86,E2 -12201.86} C_VEL
LIN {X 0,Y 376.008,Z 273.675,A -85,B 0,C 180,E1 -12203.267,E2 -12203.267} C_VEL
LIN {X 0,Y 376.431,Z 268.502,A -85,B 0,C 180,E1 -12204.356,E2 -12204.356} C_VEL
LIN {X 0,Y 377.076,Z 261.507,A -85,B 0,C 180,E1 -12205.551,E2 -12205.551} C_VEL
LIN {X 0,Y 377.84,Z 252.849,A -85,B 0,C 180,E1 -12206.715,E2 -12206.715} C_VEL
LIN {X 0,Y 378.315,Z 244.876,A -85,B 0,C 180,E1 -12207.562,E2 -12207.562} C_VEL
LIN {X 0,Y 378.84,Z 236.886,A -85,B 0,C 180,E1 -12208.239,E2 -12208.239} C_VEL
LIN {X 0,Y 377.395,Z 228.057,A -85,B 0,C 180,E1 -12208.917,E2 -12208.917} C_VEL
LIN {X 0,Y 375.123,Z 218.036,A -85,B 0,C 180,E1 -12209.544,E2 -12209.544} C_VEL
LIN {X 0,Y 374.97,Z 217.079,A -85,B 0,C 180,E1 -12209.6,E2 -12209.6} C_VEL
LIN {X 0,Y 375.122,Z 213.86,A -85,B 0,C 180,E1 -12212.072,E2 -12212.072} C_VEL
LIN {X 0,Y 375.26,Z 209.274,A -85,B 0,C 180,E1 -12215.669,E2 -12215.669} C_VEL
LIN {X 0,Y 375.463,Z 206.33,A -85,B 0,C 180,E1 -12218.016,E2 -12218.016} C_VEL
LIN {X 0,Y 375.697,Z 202.136,A -85,B 0,C 180,E1 -12221.458,E2 -12221.458} C_VEL
LIN {X 0,Y 375.958,Z 198.102,A -85,B 0,C 180,E1 -12224.83,E2 -12224.83} C_VEL
LIN {X 0,Y 376.098,Z 195.564,A -85,B 0,C 180,E1 -12227.043,E2 -12227.043} C_VEL
LIN {X 0,Y 376,Z 194.468,A -85,B 0,C 180,E1 -12228.136,E2 -12228.136} C_VEL
LIN {X 0,Y 376.278,Z 194.433,A -85,B 0,C 180,E1 -12231.857,E2 -12231.857} C_VEL
LIN {X 0,Y 376.172,Z 194.447,A -85,B 0,C 180,E1 -12234.641,E2 -12234.641} C_VEL
LIN {X 0,Y 376.353,Z 194.42,A -85,B 0,C 180,E1 -12237.861,E2 -12237.861} C_VEL
LIN {X 0,Y 376.49,Z 194.402,A -85,B 0,C 180,E1 -12240.001,E2 -12240.001} C_VEL
LIN {X 0,Y 376.186,Z 194.437,A -85,B 0,C 180,E1 -12243.214,E2 -12243.214} C_VEL
LIN {X 0,Y 376.234,Z 194.433,A -85,B 0,C 180,E1 -12246.436,E2 -12246.436} C_VEL
LIN {X 0,Y 376.115,Z 194.449,A -85,B 0,C 180,E1 -12249.682,E2 -12249.682} C_VEL
LIN {X 0,Y 376.091,Z 194.452,A -85,B 0,C 180,E1 -12253.658,E2 -12253.658} C_VEL
LIN {X 0,Y 376.046,Z 194.457,A -85,B 0,C 180,E1 -12257.608,E2 -12257.608} C_VEL
LIN {X 0,Y 375.98,Z 194.466,A -85,B 0,C 180,E1 -12260.833,E2 -12260.833} C_VEL
LIN {X 0,Y 375.996,Z 194.464,A -85,B 0,C 180,E1 -12264.282,E2 -12264.282} C_VEL
LIN {X 0,Y 376.022,Z 194.462,A -85,B 0,C 180,E1 -12266.653,E2 -12266.653} C_VEL
LIN {X 0,Y 375.967,Z 194.467,A -85,B 0,C 180,E1 -12270.313,E2 -12270.313} C_VEL
LIN {X 0,Y 375.962,Z 194.466,A -85,B 0,C 180,E1 -12274.112,E2 -12274.112} C_VEL
LIN {X 0,Y 375.955,Z 194.469,A -85,B 0,C 180,E1 -12276.742,E2 -12276.742} C_VEL
LIN {X 0,Y 375.99,Z 194.466,A -85,B 0,C 180,E1 -12279.971,E2 -12279.971} C_VEL
LIN {X 0,Y 375.932,Z 194.475,A -85,B 0,C 180,E1 -12283.766,E2 -12283.766} C_VEL
LIN {X 0,Y 375.936,Z 194.474,A -85,B 0,C 180,E1 -12286.811,E2 -12286.811} C_VEL
LIN {X 0,Y 375.999,Z 194.464,A -85,B 0,C 180,E1 -12290.542,E2 -12290.542} C_VEL
LIN {X 0,Y 376.04,Z 194.695,A -85,B 0,C 180,E1 -12291.015,E2 -12291.015} C_VEL
LIN {X 0,Y 377.148,Z 200.609,A -85,B 0,C 180,E1 -12294.713,E2 -12294.713} C_VEL
LIN {X 0,Y 378.094,Z 206.407,A -85,B 0,C 180,E1 -12298.011,E2 -12298.011} C_VEL
LIN {X 0,Y 377.62,Z 211.194,A -85,B 0,C 180,E1 -12300.449,E2 -12300.449} C_VEL
LIN {X 0,Y 376.738,Z 218.646,A -85,B 0,C 180,E1 -12304.06,E2 -12304.06} C_VEL
LIN {X 0,Y 376.032,Z 225.967,A -85,B 0,C 180,E1 -12307.472,E2 -12307.472} C_VEL
LIN {X 0,Y 375.488,Z 233.571,A -85,B 0,C 180,E1 -12310.88,E2 -12310.88} C_VEL
LIN {X 0,Y 375.024,Z 242.03,A -85,B 0,C 180,E1 -12314.581,E2 -12314.581} C_VEL
LIN {X 0,Y 376.946,Z 255.202,A -85,B 0,C 180,E1 -12315.242,E2 -12315.242} C_VEL
LIN {X 0,Y 377.782,Z 264.827,A -85,B 0,C 180,E1 -12315.892,E2 -12315.892} C_VEL
LIN {X 0,Y 377.957,Z 271.478,A -85,B 0,C 180,E1 -12316.423,E2 -12316.423} C_VEL
LIN {X 0,Y 377.389,Z 279.914,A -85,B 0,C 180,E1 -12317.224,E2 -12317.224} C_VEL
LIN {X 0,Y 376.679,Z 287.9,A -85,B 0,C 180,E1 -12318.157,E2 -12318.157} C_VEL
LIN {X 0,Y 376.26,Z 293.662,A -85,B 0,C 180,E1 -12318.962,E2 -12318.962} C_VEL
LIN {X 0,Y 375.695,Z 300.101,A -85,B 0,C 180,E1 -12320.036,E2 -12320.036} C_VEL
LIN {X 0,Y 375.219,Z 306.649,A -85,B 0,C 180,E1 -12321.382,E2 -12321.382} C_VEL
LIN {X 0,Y 374.921,Z 310.91,A -85,B 0,C 180,E1 -12322.46,E2 -12322.46} C_VEL
LIN {X 0,Y 374.717,Z 314.444,A -85,B 0,C 180,E1 -12323.539,E2 -12323.539} C_VEL
LIN {X 0,Y 374.61,Z 318.524,A -85,B 0,C 180,E1 -12325.157,E2 -12325.157} C_VEL
LIN {X 0,Y 374.511,Z 321.336,A -85,B 0,C 180,E1 -12326.773,E2 -12326.773} C_VEL
LIN {X 0,Y 374.556,Z 322.464,A -85,B 0,C 180,E1 -12327.85,E2 -12327.85} C_VEL
LIN {X 0,Y 374.623,Z 323.106,A -85,B 0,C 180,E1 -12328.925,E2 -12328.925} C_VEL
LIN {X 0,Y 374.61,Z 323.265,A -85,B 0,C 180,E1 -12330,E2 -12330} C_VEL
LIN {X 0,Y 374.625,Z 322.933,A -85,B 0,C 180,E1 -12331.075,E2 -12331.075} C_VEL
LIN {X 0,Y 374.578,Z 322,A -85,B 0,C 180,E1 -12332.151,E2 -12332.151} C_VEL
LIN {X 0,Y 374.526,Z 320.527,A -85,B 0,C 180,E1 -12333.227,E2 -12333.227} C_VEL
LIN {X 0,Y 374.627,Z 317.379,A -85,B 0,C 180,E1 -12334.843,E2 -12334.843} C_VEL
LIN {X 0,Y 374.717,Z 312.762,A -85,B 0,C 180,E1 -12336.462,E2 -12336.462} C_VEL
LIN {X 0,Y 374.958,Z 307.671,A -85,B 0,C 180,E1 -12337.81,E2 -12337.81} C_VEL
LIN {X 0,Y 375.239,Z 302.685,A -85,B 0,C 180,E1 -12338.889,E2 -12338.889} C_VEL
LIN {X 0,Y 375.602,Z 296.663,A -85,B 0,C 180,E1 -12339.967,E2 -12339.967} C_VEL
LIN {X 0,Y 376.075,Z 289.325,A -85,B 0,C 180,E1 -12341.043,E2 -12341.043} C_VEL
LIN {X 0,Y 376.575,Z 281.47,A -85,B 0,C 180,E1 -12341.983,E2 -12341.983} C_VEL
LIN {X 0,Y 377.124,Z 273.187,A -85,B 0,C 180,E1 -12342.786,E2 -12342.786} C_VEL
LIN {X 0,Y 377.076,Z 265.487,A -85,B 0,C 180,E1 -12343.397,E2 -12343.397} C_VEL
LIN {X 0,Y 376.073,Z 253.993,A -85,B 0,C 180,E1 -12344.129,E2 -12344.129} C_VEL
LIN {X 0,Y 374.918,Z 242.893,A -85,B 0,C 180,E1 -12344.624,E2 -12344.624} C_VEL
LIN {X 0,Y 375.358,Z 233.773,A -85,B 0,C 180,E1 -12348.56,E2 -12348.56} C_VEL
LIN {X 0,Y 375.82,Z 226.02,A -85,B 0,C 180,E1 -12351.963,E2 -12351.963} C_VEL
LIN {X 0,Y 376.463,Z 218.266,A -85,B 0,C 180,E1 -12355.428,E2 -12355.428} C_VEL
LIN {X 0,Y 377.258,Z 210.486,A -85,B 0,C 180,E1 -12358.971,E2 -12358.971} C_VEL
LIN {X 0,Y 377.751,Z 205.311,A -85,B 0,C 180,E1 -12361.395,E2 -12361.395} C_VEL
LIN {X 0,Y 377.041,Z 200.092,A -85,B 0,C 180,E1 -12364.001,E2 -12364.001} C_VEL
LIN {X 0,Y 375.998,Z 194.464,A -85,B 0,C 180,E1 -12366.987,E2 -12366.987} C_VEL
LIN {X 0,Y 375.992,Z 194.463,A -85,B 0,C 180,E1 -12369.97,E2 -12369.97} C_VEL
LIN {X 0,Y 375.933,Z 194.468,A -85,B 0,C 180,E1 -12373.766,E2 -12373.766} C_VEL
LIN {X 0,Y 375.938,Z 194.469,A -85,B 0,C 180,E1 -12376.81,E2 -12376.81} C_VEL
LIN {X 0,Y 375.945,Z 194.469,A -85,B 0,C 180,E1 -12380.535,E2 -12380.535} C_VEL
LIN {X 0,Y 375.967,Z 194.465,A -85,B 0,C 180,E1 -12383.495,E2 -12383.495} C_VEL
LIN {X 0,Y 375.965,Z 194.468,A -85,B 0,C 180,E1 -12385.888,E2 -12385.888} C_VEL
LIN {X 0,Y 375.969,Z 194.466,A -85,B 0,C 180,E1 -12389.687,E2 -12389.687} C_VEL
LIN {X 0,Y 376.024,Z 194.458,A -85,B 0,C 180,E1 -12393.348,E2 -12393.348} C_VEL
LIN {X 0,Y 375.983,Z 194.461,A -85,B 0,C 180,E1 -12396.887,E2 -12396.887} C_VEL
LIN {X 0,Y 376.002,Z 194.46,A -85,B 0,C 180,E1 -12400.339,E2 -12400.339} C_VEL
LIN {X 0,Y 376.034,Z 194.459,A -85,B 0,C 180,E1 -12403.718,E2 -12403.718} C_VEL
LIN {X 0,Y 376.108,Z 194.448,A -85,B 0,C 180,E1 -12407.041,E2 -12407.041} C_VEL
LIN {X 0,Y 376.117,Z 194.445,A -85,B 0,C 180,E1 -12410.318,E2 -12410.318} C_VEL
LIN {X 0,Y 376.232,Z 194.434,A -85,B 0,C 180,E1 -12413.564,E2 -12413.564} C_VEL
LIN {X 0,Y 376.354,Z 194.416,A -85,B 0,C 180,E1 -12417.859,E2 -12417.859} C_VEL
LIN {X 0,Y 376.489,Z 194.399,A -85,B 0,C 180,E1 -12419.999,E2 -12419.999} C_VEL
LIN {X 0,Y 376.187,Z 194.44,A -85,B 0,C 180,E1 -12423.212,E2 -12423.212} C_VEL
LIN {X 0,Y 376.214,Z 194.433,A -85,B 0,C 180,E1 -12426.616,E2 -12426.616} C_VEL
LIN {X 0,Y 376.115,Z 194.445,A -85,B 0,C 180,E1 -12429.681,E2 -12429.681} C_VEL
LIN {X 0,Y 376.091,Z 194.448,A -85,B 0,C 180,E1 -12433.657,E2 -12433.657} C_VEL
LIN {X 0,Y 376.033,Z 194.456,A -85,B 0,C 180,E1 -12437.399,E2 -12437.399} C_VEL
LIN {X 0,Y 375.978,Z 194.466,A -85,B 0,C 180,E1 -12440.831,E2 -12440.831} C_VEL
LIN {X 0,Y 375.988,Z 194.464,A -85,B 0,C 180,E1 -12444.281,E2 -12444.281} C_VEL
LIN {X 0,Y 376.019,Z 194.461,A -85,B 0,C 180,E1 -12446.651,E2 -12446.651} C_VEL
LIN {X 0,Y 375.969,Z 194.464,A -85,B 0,C 180,E1 -12449.078,E2 -12449.078} C_VEL
LIN {X 0,Y 375.949,Z 194.467,A -85,B 0,C 180,E1 -12452.827,E2 -12452.827} C_VEL
LIN {X 0,Y 375.956,Z 194.465,A -85,B 0,C 180,E1 -12455.414,E2 -12455.414} C_VEL
LIN {X 0,Y 375.972,Z 194.468,A -85,B 0,C 180,E1 -12458.269,E2 -12458.269} C_VEL
LIN {X 0,Y 375.93,Z 194.47,A -85,B 0,C 180,E1 -12461.6,E2 -12461.6} C_VEL
LIN {X 0,Y 375.922,Z 194.47,A -85,B 0,C 180,E1 -12465.267,E2 -12465.267} C_VEL
LIN {X 0,Y 375.929,Z 194.47,A -85,B 0,C 180,E1 -12468.398,E2 -12468.398} C_VEL
LIN {X 0,Y 375.97,Z 194.467,A -85,B 0,C 180,E1 -12471.728,E2 -12471.728} C_VEL
LIN {X 0,Y 375.974,Z 194.465,A -85,B 0,C 180,E1 -12475.332,E2 -12475.332} C_VEL
LIN {X 0,Y 375.954,Z 194.465,A -85,B 0,C 180,E1 -12478.437,E2 -12478.437} C_VEL
LIN {X 0,Y 375.995,Z 194.461,A -85,B 0,C 180,E1 -12482.141,E2 -12482.141} C_VEL
LIN {X 0,Y 375.999,Z 194.46,A -85,B 0,C 180,E1 -12484.538,E2 -12484.538} C_VEL
LIN {X 0,Y 375.956,Z 194.465,A -85,B 0,C 180,E1 -12488.045,E2 -12488.045} C_VEL
LIN {X 0,Y 376.016,Z 194.461,A -85,B 0,C 180,E1 -12491.473,E2 -12491.473} C_VEL
LIN {X 0,Y 376.052,Z 194.456,A -85,B 0,C 180,E1 -12494.832,E2 -12494.832} C_VEL
LIN {X 0,Y 376.051,Z 194.453,A -85,B 0,C 180,E1 -12498.136,E2 -12498.136} C_VEL
LIN {X 0,Y 376.249,Z 194.429,A -85,B 0,C 180,E1 -12501.877,E2 -12501.877} C_VEL
LIN {X 0,Y 376.163,Z 194.443,A -85,B 0,C 180,E1 -12504.64,E2 -12504.64} C_VEL
LIN {X 0,Y 376.343,Z 194.417,A -85,B 0,C 180,E1 -12507.859,E2 -12507.859} C_VEL
LIN {X 0,Y 376.479,Z 194.4,A -85,B 0,C 180,E1 -12510,E2 -12510} C_VEL
LIN {X 0,Y 376.181,Z 194.438,A -85,B 0,C 180,E1 -12513.213,E2 -12513.213} C_VEL
LIN {X 0,Y 376.238,Z 194.434,A -85,B 0,C 180,E1 -12516.435,E2 -12516.435} C_VEL
LIN {X 0,Y 376.196,Z 194.439,A -85,B 0,C 180,E1 -12518.595,E2 -12518.595} C_VEL
LIN {X 0,Y 375.998,Z 194.461,A -85,B 0,C 180,E1 -12521.865,E2 -12521.865} C_VEL
LIN {X 0,Y 375.846,Z 194.482,A -85,B 0,C 180,E1 -12524.069,E2 -12524.069} C_VEL
LIN {X 0,Y 375.631,Z 194.731,A -85,B 0,C 180,E1 -12525.463,E2 -12525.463} C_VEL
LIN {X 0,Y 375.373,Z 198.736,A -85,B 0,C 180,E1 -12528.559,E2 -12528.559} C_VEL
LIN {X 0,Y 375.211,Z 203.269,A -85,B 0,C 180,E1 -12532,E2 -12532} C_VEL
LIN {X 0,Y 375.023,Z 208.549,A -85,B 0,C 180,E1 -12535.907,E2 -12535.907} C_VEL
LIN {X 0,Y 374.827,Z 213.041,A -85,B 0,C 180,E1 -12539.176,E2 -12539.176} C_VEL
LIN {X 0,Y 374.809,Z 216.041,A -85,B 0,C 180,E1 -12541.355,E2 -12541.355} C_VEL
LIN {X 0,Y 376.65,Z 227.307,A -85,B 0,C 180,E1 -12541.969,E2 -12541.969} C_VEL
LIN {X 0,Y 377.789,Z 235.796,A -85,B 0,C 180,E1 -12542.569,E2 -12542.569} C_VEL
LIN {X 0,Y 377.3,Z 245.333,A -85,B 0,C 180,E1 -12543.373,E2 -12543.373} C_VEL
LIN {X 0,Y 376.773,Z 254.613,A -85,B 0,C 180,E1 -12544.404,E2 -12544.404} C_VEL
LIN {X 0,Y 376.283,Z 261.638,A -85,B 0,C 180,E1 -12545.38,E2 -12545.38} C_VEL
LIN {X 0,Y 376.109,Z 263.882,A -85,B 0,C 180,E1 -12545.731,E2 -12545.731} C_VEL
LIN {X 0,Y 375.192,Z 267.833,A -85,B 0,C 180,E1 -12546.388,E2 -12546.388} C_VEL
LIN {X 0,Y 371.959,Z 273.629,A -85,B 0,C 180,E1 -12547.52,E2 -12547.52} C_VEL
LIN {X 0,Y 368.738,Z 278.589,A -85,B 0,C 180,E1 -12548.762,E2 -12548.762} C_VEL
LIN {X 0,Y 367.858,Z 281.149,A -85,B 0,C 180,E1 -12549.581,E2 -12549.581} C_VEL
LIN {X 0,Y 367.602,Z 285.012,A -85,B 0,C 180,E1 -12551.154,E2 -12551.154} C_VEL
LIN {X 0,Y 367.518,Z 286.558,A -85,B 0,C 180,E1 -12552.013,E2 -12552.013} C_VEL
LIN {X 0,Y 367.384,Z 288.438,A -85,B 0,C 180,E1 -12553.525,E2 -12553.525} C_VEL
LIN {X 0,Y 367.33,Z 289.302,A -85,B 0,C 180,E1 -12555.065,E2 -12555.065} C_VEL
LIN {X 0,Y 367.421,Z 289.112,A -85,B 0,C 180,E1 -12556.624,E2 -12556.624} C_VEL
LIN {X 0,Y 367.617,Z 287.742,A -85,B 0,C 180,E1 -12558.21,E2 -12558.21} C_VEL
LIN {X 0,Y 367.912,Z 285.094,A -85,B 0,C 180,E1 -12559.827,E2 -12559.827} C_VEL
LIN {X 0,Y 368.332,Z 281.094,A -85,B 0,C 180,E1 -12561.472,E2 -12561.472} C_VEL
LIN {X 0,Y 368.916,Z 275.405,A -85,B 0,C 180,E1 -12563.141,E2 -12563.141} C_VEL
LIN {X 0,Y 369.41,Z 269.827,A -85,B 0,C 180,E1 -12564.387,E2 -12564.387} C_VEL
LIN {X 0,Y 369.967,Z 264.145,A -85,B 0,C 180,E1 -12565.424,E2 -12565.424} C_VEL
LIN {X 0,Y 370.474,Z 258.464,A -85,B 0,C 180,E1 -12566.294,E2 -12566.294} C_VEL
LIN {X 0,Y 371.111,Z 251.522,A -85,B 0,C 180,E1 -12567.175,E2 -12567.175} C_VEL
LIN {X 0,Y 371.662,Z 243.266,A -85,B 0,C 180,E1 -12568.032,E2 -12568.032} C_VEL
LIN {X 0,Y 371.931,Z 237.556,A -85,B 0,C 180,E1 -12568.523,E2 -12568.523} C_VEL
LIN {X 0,Y 370.541,Z 229.139,A -85,B 0,C 180,E1 -12569.197,E2 -12569.197} C_VEL
LIN {X 0,Y 368.497,Z 219.928,A -85,B 0,C 180,E1 -12569.801,E2 -12569.801} C_VEL
LIN {X 0,Y 367.914,Z 217.339,A -85,B 0,C 180,E1 -12569.985,E2 -12569.985} C_VEL
LIN {X 0,Y 368.083,Z 213.836,A -85,B 0,C 180,E1 -12572.727,E2 -12572.727} C_VEL
LIN {X 0,Y 368.294,Z 209.288,A -85,B 0,C 180,E1 -12576.377,E2 -12576.377} C_VEL
LIN {X 0,Y 368.537,Z 204.968,A -85,B 0,C 180,E1 -12579.926,E2 -12579.926} C_VEL
LIN {X 0,Y 368.825,Z 200.859,A -85,B 0,C 180,E1 -12583.393,E2 -12583.393} C_VEL
LIN {X 0,Y 369.091,Z 196.984,A -85,B 0,C 180,E1 -12586.793,E2 -12586.793} C_VEL
LIN {X 0,Y 368.991,Z 195.768,A -85,B 0,C 180,E1 -12587.907,E2 -12587.907} C_VEL
LIN {X 0,Y 369,Z 195.337,A -85,B 0,C 180,E1 -12589.021,E2 -12589.021} C_VEL
LIN {X 0,Y 369.194,Z 195.316,A -85,B 0,C 180,E1 -12592.343,E2 -12592.343} C_VEL
LIN {X 0,Y 369.145,Z 195.322,A -85,B 0,C 180,E1 -12594.539,E2 -12594.539} C_VEL
LIN {X 0,Y 369.318,Z 195.297,A -85,B 0,C 180,E1 -12597.82,E2 -12597.82} C_VEL
LIN {X 0,Y 369.46,Z 195.278,A -85,B 0,C 180,E1 -12600.001,E2 -12600.001} C_VEL
LIN {X 0,Y 369.318,Z 195.296,A -85,B 0,C 180,E1 -12602.182,E2 -12602.182} C_VEL
LIN {X 0,Y 369.193,Z 195.311,A -85,B 0,C 180,E1 -12606.559,E2 -12606.559} C_VEL
LIN {X 0,Y 369.065,Z 195.326,A -85,B 0,C 180,E1 -12609.869,E2 -12609.869} C_VEL
LIN {X 0,Y 369.039,Z 195.331,A -85,B 0,C 180,E1 -12613.773,E2 -12613.773} C_VEL
LIN {X 0,Y 369.003,Z 195.334,A -85,B 0,C 180,E1 -12617.769,E2 -12617.769} C_VEL
LIN {X 0,Y 368.931,Z 195.343,A -85,B 0,C 180,E1 -12621.22,E2 -12621.22} C_VEL
LIN {X 0,Y 368.96,Z 195.338,A -85,B 0,C 180,E1 -12624.776,E2 -12624.776} C_VEL
LIN {X 0,Y 368.965,Z 195.339,A -85,B 0,C 180,E1 -12627.204,E2 -12627.204} C_VEL
LIN {X 0,Y 368.921,Z 195.345,A -85,B 0,C 180,E1 -12629.691,E2 -12629.691} C_VEL
LIN {X 0,Y 368.899,Z 195.346,A -85,B 0,C 180,E1 -12633.044,E2 -12633.044} C_VEL
LIN {X 0,Y 368.919,Z 195.344,A -85,B 0,C 180,E1 -12636.197,E2 -12636.197} C_VEL
LIN {X 0,Y 368.904,Z 195.348,A -85,B 0,C 180,E1 -12638.954,E2 -12638.954} C_VEL
LIN {X 0,Y 368.883,Z 195.352,A -85,B 0,C 180,E1 -12642.01,E2 -12642.01} C_VEL
LIN {X 0,Y 368.882,Z 195.353,A -85,B 0,C 180,E1 -12645.176,E2 -12645.176} C_VEL
LIN {X 0,Y 368.885,Z 195.352,A -85,B 0,C 180,E1 -12648.178,E2 -12648.178} C_VEL
LIN {X 0,Y 368.989,Z 195.54,A -85,B 0,C 180,E1 -12650.53,E2 -12650.53} C_VEL
LIN {X 0,Y 369.952,Z 200.751,A -85,B 0,C 180,E1 -12653.921,E2 -12653.921} C_VEL
LIN {X 0,Y 370.955,Z 206.504,A -85,B 0,C 180,E1 -12657.32,E2 -12657.32} C_VEL
LIN {X 0,Y 371.1,Z 208.551,A -85,B 0,C 180,E1 -12658.455,E2 -12658.455} C_VEL
LIN {X 0,Y 370.306,Z 214.828,A -85,B 0,C 180,E1 -12661.675,E2 -12661.675} C_VEL
LIN {X 0,Y 369.458,Z 222.165,A -85,B 0,C 180,E1 -12665.261,E2 -12665.261} C_VEL
LIN {X 0,Y 368.723,Z 230.274,A -85,B 0,C 180,E1 -12669.062,E2 -12669.062} C_VEL
LIN {X 0,Y 368.16,Z 238.21,A -85,B 0,C 180,E1 -12672.646,E2 -12672.646} C_VEL
LIN {X 0,Y 367.988,Z 241.708,A -85,B 0,C 180,E1 -12674.208,E2 -12674.208} C_VEL
LIN {X 0,Y 369.962,Z 254.79,A -85,B 0,C 180,E1 -12674.904,E2 -12674.904} C_VEL
LIN {X 0,Y 370.81,Z 263.844,A -85,B 0,C 180,E1 -12675.527,E2 -12675.527} C_VEL
LIN {X 0,Y 371.06,Z 271.606,A -85,B 0,C 180,E1 -12676.165,E2 -12676.165} C_VEL
LIN {X 0,Y 370.484,Z 279.961,A -85,B 0,C 180,E1 -12676.982,E2 -12676.982} C_VEL
LIN {X 0,Y 369.711,Z 287.886,A -85,B 0,C 180,E1 -12677.93,E2 -12677.93} C_VEL
LIN {X 0,Y 369.141,Z 295.309,A -85,B 0,C 180,E1 -12679.025,E2 -12679.025} C_VEL
LIN {X 0,Y 368.498,Z 302.856,A -85,B 0,C 180,E1 -12680.394,E2 -12680.394} C_VEL
LIN {X 0,Y 368.016,Z 308.79,A -85,B 0,C 180,E1 -12681.766,E2 -12681.766} C_VEL
LIN {X 0,Y 367.778,Z 312.656,A -85,B 0,C 180,E1 -12682.865,E2 -12682.865} C_VEL
LIN {X 0,Y 367.503,Z 317.104,A -85,B 0,C 180,E1 -12684.513,E2 -12684.513} C_VEL
LIN {X 0,Y 367.51,Z 319.395,A -85,B 0,C 180,E1 -12685.613,E2 -12685.613} C_VEL
LIN {X 0,Y 367.427,Z 321.071,A -85,B 0,C 180,E1 -12686.711,E2 -12686.711} C_VEL
LIN {X 0,Y 367.456,Z 322.172,A -85,B 0,C 180,E1 -12687.808,E2 -12687.808} C_VEL
LIN {X 0,Y 367.538,Z 322.79,A -85,B 0,C 180,E1 -12688.905,E2 -12688.905} C_VEL
LIN {X 0,Y 367.544,Z 322.926,A -85,B 0,C 180,E1 -12690,E2 -12690} C_VEL
LIN {X 0,Y 367.558,Z 322.576,A -85,B 0,C 180,E1 -12691.096,E2 -12691.096} C_VEL
LIN {X 0,Y 367.479,Z 321.635,A -85,B 0,C 180,E1 -12692.192,E2 -12692.192} C_VEL
LIN {X 0,Y 367.477,Z 319.261,A -85,B 0,C 180,E1 -12693.838,E2 -12693.838} C_VEL
LIN {X 0,Y 367.507,Z 315.512,A -85,B 0,C 180,E1 -12695.487,E2 -12695.487} C_VEL
LIN {X 0,Y 367.647,Z 312.28,A -85,B 0,C 180,E1 -12696.586,E2 -12696.586} C_VEL
LIN {X 0,Y 367.903,Z 307.151,A -85,B 0,C 180,E1 -12697.961,E2 -12697.961} C_VEL
LIN {X 0,Y 368.188,Z 302.12,A -85,B 0,C 180,E1 -12699.061,E2 -12699.061} C_VEL
LIN {X 0,Y 368.562,Z 296.045,A -85,B 0,C 180,E1 -12700.16,E2 -12700.16} C_VEL
LIN {X 0,Y 369.077,Z 288.646,A -85,B 0,C 180,E1 -12701.256,E2 -12701.256} C_VEL
LIN {X 0,Y 369.61,Z 280.716,A -85,B 0,C 180,E1 -12702.213,E2 -12702.213} C_VEL
LIN {X 0,Y 370.189,Z 270.818,A -85,B 0,C 180,E1 -12703.169,E2 -12703.169} C_VEL
LIN {X 0,Y 369.582,Z 259.834,A -85,B 0,C 180,E1 -12703.977,E2 -12703.977} C_VEL
LIN {X 0,Y 368.608,Z 249.931,A -85,B 0,C 180,E1 -12704.528,E2 -12704.528} C_VEL
LIN {X 0,Y 367.817,Z 242.659,A -85,B 0,C 180,E1 -12704.842,E2 -12704.842} C_VEL
LIN {X 0,Y 368.257,Z 234.714,A -85,B 0,C 180,E1 -12708.355,E2 -12708.355} C_VEL
LIN {X 0,Y 368.828,Z 225.696,A -85,B 0,C 180,E1 -12712.402,E2 -12712.402} C_VEL
LIN {X 0,Y 369.515,Z 217.935,A -85,B 0,C 180,E1 -12715.942,E2 -12715.942} C_VEL
LIN {X 0,Y 370.337,Z 210.202,A -85,B 0,C 180,E1 -12719.565,E2 -12719.565} C_VEL
LIN {X 0,Y 370.728,Z 206.27,A -85,B 0,C 180,E1 -12721.451,E2 -12721.451} C_VEL
LIN {X 0,Y 370.025,Z 201.108,A -85,B 0,C 180,E1 -12724.077,E2 -12724.077} C_VEL
LIN {X 0,Y 368.951,Z 195.342,A -85,B 0,C 180,E1 -12727.267,E2 -12727.267} C_VEL
LIN {X 0,Y 368.914,Z 195.346,A -85,B 0,C 180,E1 -12730.37,E2 -12730.37} C_VEL
LIN {X 0,Y 368.886,Z 195.345,A -85,B 0,C 180,E1 -12733.616,E2 -12733.616} C_VEL
LIN {X 0,Y 368.889,Z 195.348,A -85,B 0,C 180,E1 -12736.696,E2 -12736.696} C_VEL
LIN {X 0,Y 368.911,Z 195.343,A -85,B 0,C 180,E1 -12739.644,E2 -12739.644} C_VEL
LIN {X 0,Y 368.904,Z 195.343,A -85,B 0,C 180,E1 -12743.144,E2 -12743.144} C_VEL
LIN {X 0,Y 368.901,Z 195.346,A -85,B 0,C 180,E1 -12746.462,E2 -12746.462} C_VEL
LIN {X 0,Y 368.934,Z 195.339,A -85,B 0,C 180,E1 -12749.046,E2 -12749.046} C_VEL
LIN {X 0,Y 368.968,Z 195.335,A -85,B 0,C 180,E1 -12752.796,E2 -12752.796} C_VEL
LIN {X 0,Y 368.938,Z 195.342,A -85,B 0,C 180,E1 -12756.116,E2 -12756.116} C_VEL
LIN {X 0,Y 368.941,Z 195.342,A -85,B 0,C 180,E1 -12759.947,E2 -12759.947} C_VEL
LIN {X 0,Y 368.981,Z 195.337,A -85,B 0,C 180,E1 -12763.398,E2 -12763.398} C_VEL
LIN {X 0,Y 369.062,Z 195.324,A -85,B 0,C 180,E1 -12766.79,E2 -12766.79} C_VEL
LIN {X 0,Y 369.067,Z 195.323,A -85,B 0,C 180,E1 -12770.131,E2 -12770.131} C_VEL
LIN {X 0,Y 369.191,Z 195.312,A -85,B 0,C 180,E1 -12773.441,E2 -12773.441} C_VEL
LIN {X 0,Y 369.319,Z 195.292,A -85,B 0,C 180,E1 -12777.818,E2 -12777.818} C_VEL
LIN {X 0,Y 369.458,Z 195.275,A -85,B 0,C 180,E1 -12779.999,E2 -12779.999} C_VEL
LIN {X 0,Y 369.32,Z 195.291,A -85,B 0,C 180,E1 -12782.18,E2 -12782.18} C_VEL
LIN {X 0,Y 369.186,Z 195.309,A -85,B 0,C 180,E1 -12786.599,E2 -12786.599} C_VEL
LIN {X 0,Y 369.065,Z 195.323,A -85,B 0,C 180,E1 -12789.867,E2 -12789.867} C_VEL
LIN {X 0,Y 369.039,Z 195.326,A -85,B 0,C 180,E1 -12793.771,E2 -12793.771} C_VEL
LIN {X 0,Y 368.991,Z 195.332,A -85,B 0,C 180,E1 -12797.742,E2 -12797.742} C_VEL
LIN {X 0,Y 368.91,Z 195.344,A -85,B 0,C 180,E1 -12801.22,E2 -12801.22} C_VEL
LIN {X 0,Y 368.954,Z 195.34,A -85,B 0,C 180,E1 -12804.774,E2 -12804.774} C_VEL
LIN {X 0,Y 368.967,Z 195.336,A -85,B 0,C 180,E1 -12807.202,E2 -12807.202} C_VEL
LIN {X 0,Y 368.917,Z 195.342,A -85,B 0,C 180,E1 -12809.689,E2 -12809.689} C_VEL
LIN {X 0,Y 368.896,Z 195.345,A -85,B 0,C 180,E1 -12813.042,E2 -12813.042} C_VEL
LIN {X 0,Y 368.915,Z 195.346,A -85,B 0,C 180,E1 -12816.195,E2 -12816.195} C_VEL
LIN {X 0,Y 368.9,Z 195.343,A -85,B 0,C 180,E1 -12818.952,E2 -12818.952} C_VEL
LIN {X 0,Y 368.878,Z 195.351,A -85,B 0,C 180,E1 -12822.008,E2 -12822.008} C_VEL
LIN {X 0,Y 368.875,Z 195.347,A -85,B 0,C 180,E1 -12825.175,E2 -12825.175} C_VEL
LIN {X 0,Y 368.878,Z 195.35,A -85,B 0,C 180,E1 -12828.176,E2 -12828.176} C_VEL
LIN {X 0,Y 368.904,Z 195.345,A -85,B 0,C 180,E1 -12831.358,E2 -12831.358} C_VEL
LIN {X 0,Y 368.931,Z 195.341,A -85,B 0,C 180,E1 -12835.146,E2 -12835.146} C_VEL
LIN {X 0,Y 368.923,Z 195.342,A -85,B 0,C 180,E1 -12839.046,E2 -12839.046} C_VEL
LIN {X 0,Y 368.98,Z 195.338,A -85,B 0,C 180,E1 -12841.564,E2 -12841.564} C_VEL
LIN {X 0,Y 368.95,Z 195.341,A -85,B 0,C 180,E1 -12845.224,E2 -12845.224} C_VEL
LIN {X 0,Y 368.93,Z 195.343,A -85,B 0,C 180,E1 -12848.973,E2 -12848.973} C_VEL
LIN {X 0,Y 368.982,Z 195.333,A -85,B 0,C 180,E1 -12852.257,E2 -12852.257} C_VEL
LIN {X 0,Y 369.029,Z 195.327,A -85,B 0,C 180,E1 -12856.227,E2 -12856.227} C_VEL
LIN {X 0,Y 369.064,Z 195.323,A -85,B 0,C 180,E1 -12860.131,E2 -12860.131} C_VEL
LIN {X 0,Y 369.179,Z 195.31,A -85,B 0,C 180,E1 -12862.342,E2 -12862.342} C_VEL
LIN {X 0,Y 369.136,Z 195.317,A -85,B 0,C 180,E1 -12864.537,E2 -12864.537} C_VEL
LIN {X 0,Y 369.308,Z 195.293,A -85,B 0,C 180,E1 -12867.819,E2 -12867.819} C_VEL
LIN {X 0,Y 369.449,Z 195.276,A -85,B 0,C 180,E1 -12870,E2 -12870} C_VEL
LIN {X 0,Y 369.31,Z 195.294,A -85,B 0,C 180,E1 -12872.181,E2 -12872.181} C_VEL
LIN {X 0,Y 369.2,Z 195.311,A -85,B 0,C 180,E1 -12876.558,E2 -12876.558} C_VEL
LIN {X 0,Y 369.128,Z 195.319,A -85,B 0,C 180,E1 -12878.761,E2 -12878.761} C_VEL
LIN {X 0,Y 368.941,Z 195.341,A -85,B 0,C 180,E1 -12882.095,E2 -12882.095} C_VEL
LIN {X 0,Y 368.695,Z 195.372,A -85,B 0,C 180,E1 -12884.912,E2 -12884.912} C_VEL
LIN {X 0,Y 368.593,Z 195.604,A -85,B 0,C 180,E1 -12885.482,E2 -12885.482} C_VEL
LIN {X 0,Y 368.292,Z 200.007,A -85,B 0,C 180,E1 -12888.929,E2 -12888.929} C_VEL
LIN {X 0,Y 368.158,Z 203.046,A -85,B 0,C 180,E1 -12891.266,E2 -12891.266} C_VEL
LIN {X 0,Y 367.989,Z 207.766,A -85,B 0,C 180,E1 -12894.845,E2 -12894.845} C_VEL
LIN {X 0,Y 367.779,Z 212.757,A -85,B 0,C 180,E1 -12898.537,E2 -12898.537} C_VEL
LIN {X 0,Y 367.735,Z 216.48,A -85,B 0,C 180,E1 -12901.145,E2 -12901.145} C_VEL
LIN {X 0,Y 369.458,Z 226.697,A -85,B 0,C 180,E1 -12901.701,E2 -12901.701} C_VEL
LIN {X 0,Y 370.768,Z 236.115,A -85,B 0,C 180,E1 -12902.377,E2 -12902.377} C_VEL
LIN {X 0,Y 370.324,Z 245.334,A -85,B 0,C 180,E1 -12903.168,E2 -12903.168} C_VEL
LIN {X 0,Y 369.747,Z 255.093,A -85,B 0,C 180,E1 -12904.27,E2 -12904.27} C_VEL
LIN {X 0,Y 369.231,Z 262.379,A -85,B 0,C 180,E1 -12905.311,E2 -12905.311} C_VEL
LIN {X 0,Y 368.735,Z 269.173,A -85,B 0,C 180,E1 -12906.507,E2 -12906.507} C_VEL
LIN {X 0,Y 368.301,Z 276.086,A -85,B 0,C 180,E1 -12908.054,E2 -12908.054} C_VEL
LIN {X 0,Y 367.858,Z 281.149,A -85,B 0,C 180,E1 -12909.581,E2 -12909.581} C_VEL
LIN {X 0,Y 367.005,Z 283.475,A -85,B 0,C 180,E1 -12910.422,E2 -12910.422} C_VEL
LIN {X 0,Y 363.941,Z 286.453,A -85,B 0,C 180,E1 -12911.823,E2 -12911.823} C_VEL
LIN {X 0,Y 360.962,Z 288.535,A -85,B 0,C 180,E1 -12913.289,E2 -12913.289} C_VEL
LIN {X 0,Y 360.256,Z 289.24,A -85,B 0,C 180,E1 -12914.217,E2 -12914.217} C_VEL
LIN {X 0,Y 360.254,Z 289.717,A -85,B 0,C 180,E1 -12915.39,E2 -12915.39} C_VEL
LIN {X 0,Y 360.355,Z 289.306,A -85,B 0,C 180,E1 -12916.954,E2 -12916.954} C_VEL
LIN {X 0,Y 360.587,Z 287.824,A -85,B 0,C 180,E1 -12918.498,E2 -12918.498} C_VEL
LIN {X 0,Y 360.864,Z 285.351,A -85,B 0,C 180,E1 -12920.009,E2 -12920.009} C_VEL
LIN {X 0,Y 361.259,Z 281.834,A -85,B 0,C 180,E1 -12921.5,E2 -12921.5} C_VEL
LIN {X 0,Y 361.806,Z 277.174,A -85,B 0,C 180,E1 -12922.976,E2 -12922.976} C_VEL
LIN {X 0,Y 362.427,Z 270.642,A -85,B 0,C 180,E1 -12924.532,E2 -12924.532} C_VEL
LIN {X 0,Y 362.974,Z 265.408,A -85,B 0,C 180,E1 -12925.531,E2 -12925.531} C_VEL
LIN {X 0,Y 363.605,Z 258.774,A -85,B 0,C 180,E1 -12926.575,E2 -12926.575} C_VEL
LIN {X 0,Y 364.307,Z 251.564,A -85,B 0,C 180,E1 -12927.502,E2 -12927.502} C_VEL
LIN {X 0,Y 364.859,Z 243.525,A -85,B 0,C 180,E1 -12928.349,E2 -12928.349} C_VEL
LIN {X 0,Y 365.195,Z 239.685,A -85,B 0,C 180,E1 -12928.696,E2 -12928.696} C_VEL
LIN {X 0,Y 363.742,Z 230.407,A -85,B 0,C 180,E1 -12929.474,E2 -12929.474} C_VEL
LIN {X 0,Y 361.714,Z 221.323,A -85,B 0,C 180,E1 -12930.101,E2 -12930.101} C_VEL
LIN {X 0,Y 360.887,Z 217.653,A -85,B 0,C 180,E1 -12930.347,E2 -12930.347} C_VEL
LIN {X 0,Y 361.069,Z 213.651,A -85,B 0,C 180,E1 -12933.555,E2 -12933.555} C_VEL
LIN {X 0,Y 361.286,Z 209.312,A -85,B 0,C 180,E1 -12937.106,E2 -12937.106} C_VEL
LIN {X 0,Y 361.569,Z 205.051,A -85,B 0,C 180,E1 -12940.706,E2 -12940.706} C_VEL
LIN {X 0,Y 361.873,Z 200.996,A -85,B 0,C 180,E1 -12944.224,E2 -12944.224} C_VEL
LIN {X 0,Y 362.068,Z 198.406,A -85,B 0,C 180,E1 -12946.532,E2 -12946.532} C_VEL
LIN {X 0,Y 361.953,Z 196.216,A -85,B 0,C 180,E1 -12948.805,E2 -12948.805} C_VEL
LIN {X 0,Y 362.157,Z 196.192,A -85,B 0,C 180,E1 -12952.194,E2 -12952.194} C_VEL
LIN {X 0,Y 362.119,Z 196.198,A -85,B 0,C 180,E1 -12954.432,E2 -12954.432} C_VEL
LIN {X 0,Y 362.282,Z 196.173,A -85,B 0,C 180,E1 -12957.777,E2 -12957.777} C_VEL
LIN {X 0,Y 362.429,Z 196.154,A -85,B 0,C 180,E1 -12960.001,E2 -12960.001} C_VEL
LIN {X 0,Y 362.282,Z 196.172,A -85,B 0,C 180,E1 -12962.224,E2 -12962.224} C_VEL
LIN {X 0,Y 362.153,Z 196.188,A -85,B 0,C 180,E1 -12966.687,E2 -12966.687} C_VEL
LIN {X 0,Y 362.002,Z 196.206,A -85,B 0,C 180,E1 -12970.064,E2 -12970.064} C_VEL
LIN {X 0,Y 362,Z 196.208,A -85,B 0,C 180,E1 -12973.9,E2 -12973.9} C_VEL
LIN {X 0,Y 361.969,Z 196.21,A -85,B 0,C 180,E1 -12977.939,E2 -12977.939} C_VEL
LIN {X 0,Y 361.894,Z 196.22,A -85,B 0,C 180,E1 -12981.654,E2 -12981.654} C_VEL
LIN {X 0,Y 361.93,Z 196.212,A -85,B 0,C 180,E1 -12985.291,E2 -12985.291} C_VEL
LIN {X 0,Y 361.916,Z 196.218,A -85,B 0,C 180,E1 -12987.779,E2 -12987.779} C_VEL
LIN {X 0,Y 361.849,Z 196.225,A -85,B 0,C 180,E1 -12991.286,E2 -12991.286} C_VEL
LIN {X 0,Y 361.856,Z 196.224,A -85,B 0,C 180,E1 -12994.281,E2 -12994.281} C_VEL
LIN {X 0,Y 361.865,Z 196.223,A -85,B 0,C 180,E1 -12997.223,E2 -12997.223} C_VEL
LIN {X 0,Y 361.838,Z 196.229,A -85,B 0,C 180,E1 -13000.756,E2 -13000.756} C_VEL
LIN {X 0,Y 361.819,Z 196.233,A -85,B 0,C 180,E1 -13004.369,E2 -13004.369} C_VEL
LIN {X 0,Y 361.838,Z 196.23,A -85,B 0,C 180,E1 -13007.568,E2 -13007.568} C_VEL
LIN {X 0,Y 361.9,Z 196.329,A -85,B 0,C 180,E1 -13009.976,E2 -13009.976} C_VEL
LIN {X 0,Y 362.741,Z 200.912,A -85,B 0,C 180,E1 -13013.086,E2 -13013.086} C_VEL
LIN {X 0,Y 363.684,Z 205.905,A -85,B 0,C 180,E1 -13016.197,E2 -13016.197} C_VEL
LIN {X 0,Y 364.121,Z 209.241,A -85,B 0,C 180,E1 -13018.132,E2 -13018.132} C_VEL
LIN {X 0,Y 363.42,Z 214.819,A -85,B 0,C 180,E1 -13021.088,E2 -13021.088} C_VEL
LIN {X 0,Y 362.505,Z 222.128,A -85,B 0,C 180,E1 -13024.753,E2 -13024.753} C_VEL
LIN {X 0,Y 361.773,Z 229.554,A -85,B 0,C 180,E1 -13028.34,E2 -13028.34} C_VEL
LIN {X 0,Y 361.171,Z 237.096,A -85,B 0,C 180,E1 -13031.86,E2 -13031.86} C_VEL
LIN {X 0,Y 360.995,Z 241.471,A -85,B 0,C 180,E1 -13033.857,E2 -13033.857} C_VEL
LIN {X 0,Y 362.893,Z 253.695,A -85,B 0,C 180,E1 -13034.496,E2 -13034.496} C_VEL
LIN {X 0,Y 363.893,Z 264.237,A -85,B 0,C 180,E1 -13035.246,E2 -13035.246} C_VEL
LIN {X 0,Y 364.15,Z 271.822,A -85,B 0,C 180,E1 -13035.898,E2 -13035.898} C_VEL
LIN {X 0,Y 363.588,Z 280.059,A -85,B 0,C 180,E1 -13036.73,E2 -13036.73} C_VEL
LIN {X 0,Y 362.761,Z 287.897,A -85,B 0,C 180,E1 -13037.696,E2 -13037.696} C_VEL
LIN {X 0,Y 362.164,Z 295.249,A -85,B 0,C 180,E1 -13038.811,E2 -13038.811} C_VEL
LIN {X 0,Y 361.474,Z 302.742,A -85,B 0,C 180,E1 -13040.205,E2 -13040.205} C_VEL
LIN {X 0,Y 360.971,Z 308.616,A -85,B 0,C 180,E1 -13041.604,E2 -13041.604} C_VEL
LIN {X 0,Y 360.712,Z 312.464,A -85,B 0,C 180,E1 -13042.724,E2 -13042.724} C_VEL
LIN {X 0,Y 360.42,Z 316.869,A -85,B 0,C 180,E1 -13044.405,E2 -13044.405} C_VEL
LIN {X 0,Y 360.422,Z 319.135,A -85,B 0,C 180,E1 -13045.527,E2 -13045.527} C_VEL
LIN {X 0,Y 360.346,Z 320.807,A -85,B 0,C 180,E1 -13046.646,E2 -13046.646} C_VEL
LIN {X 0,Y 360.356,Z 321.885,A -85,B 0,C 180,E1 -13047.765,E2 -13047.765} C_VEL
LIN {X 0,Y 360.455,Z 322.474,A -85,B 0,C 180,E1 -13048.883,E2 -13048.883} C_VEL
LIN {X 0,Y 360.479,Z 322.582,A -85,B 0,C 180,E1 -13050,E2 -13050} C_VEL
LIN {X 0,Y 360.474,Z 322.208,A -85,B 0,C 180,E1 -13051.117,E2 -13051.117} C_VEL
LIN {X 0,Y 360.381,Z 321.26,A -85,B 0,C 180,E1 -13052.236,E2 -13052.236} C_VEL
LIN {X 0,Y 360.406,Z 318.827,A -85,B 0,C 180,E1 -13053.914,E2 -13053.914} C_VEL
LIN {X 0,Y 360.452,Z 316.511,A -85,B 0,C 180,E1 -13055.034,E2 -13055.034} C_VEL
LIN {X 0,Y 360.585,Z 311.764,A -85,B 0,C 180,E1 -13056.716,E2 -13056.716} C_VEL
LIN {X 0,Y 360.825,Z 306.587,A -85,B 0,C 180,E1 -13058.118,E2 -13058.118} C_VEL
LIN {X 0,Y 361.232,Z 300.083,A -85,B 0,C 180,E1 -13059.519,E2 -13059.519} C_VEL
LIN {X 0,Y 361.811,Z 291.936,A -85,B 0,C 180,E1 -13060.917,E2 -13060.917} C_VEL
LIN {X 0,Y 362.372,Z 283.56,A -85,B 0,C 180,E1 -13062.034,E2 -13062.034} C_VEL
LIN {X 0,Y 363.073,Z 274.374,A -85,B 0,C 180,E1 -13063.005,E2 -13063.005} C_VEL
LIN {X 0,Y 363.101,Z 267.878,A -85,B 0,C 180,E1 -13063.578,E2 -13063.578} C_VEL
LIN {X 0,Y 362.494,Z 259.25,A -85,B 0,C 180,E1 -13064.21,E2 -13064.21} C_VEL
LIN {X 0,Y 361.502,Z 249.414,A -85,B 0,C 180,E1 -13064.766,E2 -13064.766} C_VEL
LIN {X 0,Y 360.771,Z 242.383,A -85,B 0,C 180,E1 -13065.103,E2 -13065.103} C_VEL
LIN {X 0,Y 361.217,Z 234.364,A -85,B 0,C 180,E1 -13068.726,E2 -13068.726} C_VEL
LIN {X 0,Y 361.724,Z 226.645,A -85,B 0,C 180,E1 -13072.264,E2 -13072.264} C_VEL
LIN {X 0,Y 362.448,Z 218.927,A -85,B 0,C 180,E1 -13075.867,E2 -13075.867} C_VEL
LIN {X 0,Y 363.265,Z 211.382,A -85,B 0,C 180,E1 -13079.47,E2 -13079.47} C_VEL
LIN {X 0,Y 363.666,Z 206.713,A -85,B 0,C 180,E1 -13081.753,E2 -13081.753} C_VEL
LIN {X 0,Y 362.771,Z 200.885,A -85,B 0,C 180,E1 -13084.821,E2 -13084.821} C_VEL
LIN {X 0,Y 361.931,Z 196.217,A -85,B 0,C 180,E1 -13087.455,E2 -13087.455} C_VEL
LIN {X 0,Y 361.831,Z 196.224,A -85,B 0,C 180,E1 -13091.331,E2 -13091.331} C_VEL
LIN {X 0,Y 361.821,Z 196.23,A -85,B 0,C 180,E1 -13094.368,E2 -13094.368} C_VEL
LIN {X 0,Y 361.836,Z 196.224,A -85,B 0,C 180,E1 -13097.569,E2 -13097.569} C_VEL
LIN {X 0,Y 361.833,Z 196.224,A -85,B 0,C 180,E1 -13100.981,E2 -13100.981} C_VEL
LIN {X 0,Y 361.878,Z 196.219,A -85,B 0,C 180,E1 -13104.655,E2 -13104.655} C_VEL
LIN {X 0,Y 361.842,Z 196.225,A -85,B 0,C 180,E1 -13108.37,E2 -13108.37} C_VEL
LIN {X 0,Y 361.913,Z 196.217,A -85,B 0,C 180,E1 -13112.221,E2 -13112.221} C_VEL
LIN {X 0,Y 361.931,Z 196.212,A -85,B 0,C 180,E1 -13114.709,E2 -13114.709} C_VEL
LIN {X 0,Y 361.866,Z 196.221,A -85,B 0,C 180,E1 -13118.345,E2 -13118.345} C_VEL
LIN {X 0,Y 361.972,Z 196.209,A -85,B 0,C 180,E1 -13122.061,E2 -13122.061} C_VEL
LIN {X 0,Y 362.002,Z 196.204,A -85,B 0,C 180,E1 -13126.1,E2 -13126.1} C_VEL
LIN {X 0,Y 362.004,Z 196.204,A -85,B 0,C 180,E1 -13129.936,E2 -13129.936} C_VEL
LIN {X 0,Y 362.152,Z 196.189,A -85,B 0,C 180,E1 -13133.313,E2 -13133.313} C_VEL
LIN {X 0,Y 362.283,Z 196.169,A -85,B 0,C 180,E1 -13137.776,E2 -13137.776} C_VEL
LIN {X 0,Y 362.428,Z 196.15,A -85,B 0,C 180,E1 -13139.999,E2 -13139.999} C_VEL
LIN {X 0,Y 362.283,Z 196.167,A -85,B 0,C 180,E1 -13142.223,E2 -13142.223} C_VEL
LIN {X 0,Y 362.151,Z 196.187,A -85,B 0,C 180,E1 -13146.686,E2 -13146.686} C_VEL
LIN {X 0,Y 362.002,Z 196.203,A -85,B 0,C 180,E1 -13150.062,E2 -13150.062} C_VEL
LIN {X 0,Y 361.999,Z 196.203,A -85,B 0,C 180,E1 -13153.898,E2 -13153.898} C_VEL
LIN {X 0,Y 361.929,Z 196.215,A -85,B 0,C 180,E1 -13156.933,E2 -13156.933} C_VEL
LIN {X 0,Y 361.887,Z 196.221,A -85,B 0,C 180,E1 -13160.46,E2 -13160.46} C_VEL
LIN {X 0,Y 361.893,Z 196.219,A -85,B 0,C 180,E1 -13164.111,E2 -13164.111} C_VEL
LIN {X 0,Y 361.942,Z 196.214,A -85,B 0,C 180,E1 -13166.72,E2 -13166.72} C_VEL
LIN {X 0,Y 361.873,Z 196.223,A -85,B 0,C 180,E1 -13170.327,E2 -13170.327} C_VEL
LIN {X 0,Y 361.853,Z 196.226,A -85,B 0,C 180,E1 -13174.279,E2 -13174.279} C_VEL
LIN {X 0,Y 361.862,Z 196.22,A -85,B 0,C 180,E1 -13177.222,E2 -13177.222} C_VEL
LIN {X 0,Y 361.832,Z 196.225,A -85,B 0,C 180,E1 -13180.754,E2 -13180.754} C_VEL
LIN {X 0,Y 361.813,Z 196.229,A -85,B 0,C 180,E1 -13184.367,E2 -13184.367} C_VEL
LIN {X 0,Y 361.831,Z 196.227,A -85,B 0,C 180,E1 -13187.567,E2 -13187.567} C_VEL
LIN {X 0,Y 361.865,Z 196.22,A -85,B 0,C 180,E1 -13190.972,E2 -13190.972} C_VEL
LIN {X 0,Y 361.869,Z 196.219,A -85,B 0,C 180,E1 -13194.654,E2 -13194.654} C_VEL
LIN {X 0,Y 361.832,Z 196.224,A -85,B 0,C 180,E1 -13198.37,E2 -13198.37} C_VEL
LIN {X 0,Y 361.896,Z 196.217,A -85,B 0,C 180,E1 -13200.954,E2 -13200.954} C_VEL
LIN {X 0,Y 361.948,Z 196.214,A -85,B 0,C 180,E1 -13203.474,E2 -13203.474} C_VEL
LIN {X 0,Y 361.883,Z 196.222,A -85,B 0,C 180,E1 -13207.144,E2 -13207.144} C_VEL
LIN {X 0,Y 361.913,Z 196.215,A -85,B 0,C 180,E1 -13210.723,E2 -13210.723} C_VEL
LIN {X 0,Y 361.939,Z 196.211,A -85,B 0,C 180,E1 -13214.226,E2 -13214.226} C_VEL
LIN {X 0,Y 361.992,Z 196.205,A -85,B 0,C 180,E1 -13216.527,E2 -13216.527} C_VEL
LIN {X 0,Y 362.028,Z 196.199,A -85,B 0,C 180,E1 -13219.938,E2 -13219.938} C_VEL
LIN {X 0,Y 362.142,Z 196.186,A -85,B 0,C 180,E1 -13222.192,E2 -13222.192} C_VEL
LIN {X 0,Y 362.11,Z 196.191,A -85,B 0,C 180,E1 -13224.431,E2 -13224.431} C_VEL
LIN {X 0,Y 362.272,Z 196.169,A -85,B 0,C 180,E1 -13227.776,E2 -13227.776} C_VEL
LIN {X 0,Y 362.419,Z 196.151,A -85,B 0,C 180,E1 -13230,E2 -13230} C_VEL
LIN {X 0,Y 362.274,Z 196.171,A -85,B 0,C 180,E1 -13232.223,E2 -13232.223} C_VEL
LIN {X 0,Y 362.164,Z 196.187,A -85,B 0,C 180,E1 -13236.686,E2 -13236.686} C_VEL
LIN {X 0,Y 362.064,Z 196.197,A -85,B 0,C 180,E1 -13238.933,E2 -13238.933} C_VEL
LIN {X 0,Y 361.886,Z 196.222,A -85,B 0,C 180,E1 -13242.335,E2 -13242.335} C_VEL
LIN {X 0,Y 361.593,Z 196.256,A -85,B 0,C 180,E1 -13245.212,E2 -13245.212} C_VEL
LIN {X 0,Y 361.276,Z 199.781,A -85,B 0,C 180,E1 -13248.135,E2 -13248.135} C_VEL
LIN {X 0,Y 361.066,Z 204.353,A -85,B 0,C 180,E1 -13251.705,E2 -13251.705} C_VEL
LIN {X 0,Y 360.872,Z 209.138,A -85,B 0,C 180,E1 -13255.369,E2 -13255.369} C_VEL
LIN {X 0,Y 360.644,Z 214.168,A -85,B 0,C 180,E1 -13259.155,E2 -13259.155} C_VEL
LIN {X 0,Y 360.65,Z 216.623,A -85,B 0,C 180,E1 -13260.906,E2 -13260.906} C_VEL
LIN {X 0,Y 362.302,Z 226.571,A -85,B 0,C 180,E1 -13261.454,E2 -13261.454} C_VEL
LIN {X 0,Y 363.628,Z 235.584,A -85,B 0,C 180,E1 -13262.107,E2 -13262.107} C_VEL
LIN {X 0,Y 363.751,Z 239.556,A -85,B 0,C 180,E1 -13262.422,E2 -13262.422} C_VEL
LIN {X 0,Y 363.242,Z 248.188,A -85,B 0,C 180,E1 -13263.252,E2 -13263.252} C_VEL
LIN {X 0,Y 362.715,Z 255.984,A -85,B 0,C 180,E1 -13264.188,E2 -13264.188} C_VEL
LIN {X 0,Y 362.226,Z 262.57,A -85,B 0,C 180,E1 -13265.15,E2 -13265.15} C_VEL
LIN {X 0,Y 361.696,Z 269.262,A -85,B 0,C 180,E1 -13266.344,E2 -13266.344} C_VEL
LIN {X 0,Y 361.294,Z 275.741,A -85,B 0,C 180,E1 -13267.79,E2 -13267.79} C_VEL
LIN {X 0,Y 360.818,Z 281.116,A -85,B 0,C 180,E1 -13269.395,E2 -13269.395} C_VEL
LIN {X 0,Y 360.549,Z 285.031,A -85,B 0,C 180,E1 -13270.982,E2 -13270.982} C_VEL
LIN {X 0,Y 360.405,Z 287.159,A -85,B 0,C 180,E1 -13272.184,E2 -13272.184} C_VEL
LIN {X 0,Y 360.282,Z 289.003,A -85,B 0,C 180,E1 -13273.802,E2 -13273.802} C_VEL
LIN {X 0,Y 360.256,Z 289.24,A -85,B 0,C 180,E1 -13274.217,E2 -13274.217} C_VEL
LIN {X 0,Y 359.587,Z 289.697,A -85,B 0,C 180,E1 -13275.151,E2 -13275.151} C_VEL
LIN {X 0,Y 356.828,Z 289.634,A -85,B 0,C 180,E1 -13276.676,E2 -13276.676} C_VEL
LIN {X 0,Y 354.565,Z 288.909,A -85,B 0,C 180,E1 -13277.903,E2 -13277.903} C_VEL
LIN {X 0,Y 353.668,Z 287.875,A -85,B 0,C 180,E1 -13278.838,E2 -13278.838} C_VEL
LIN {X 0,Y 353.635,Z 287.419,A -85,B 0,C 180,E1 -13279.15,E2 -13279.15} C_VEL
LIN {X 0,Y 353.973,Z 284.548,A -85,B 0,C 180,E1 -13280.744,E2 -13280.744} C_VEL
LIN {X 0,Y 354.551,Z 279.959,A -85,B 0,C 180,E1 -13282.456,E2 -13282.456} C_VEL
LIN {X 0,Y 355.107,Z 274.657,A -85,B 0,C 180,E1 -13283.932,E2 -13283.932} C_VEL
LIN {X 0,Y 355.757,Z 268.466,A -85,B 0,C 180,E1 -13285.292,E2 -13285.292} C_VEL
LIN {X 0,Y 356.592,Z 260.53,A -85,B 0,C 180,E1 -13286.663,E2 -13286.663} C_VEL
LIN {X 0,Y 357.421,Z 252.592,A -85,B 0,C 180,E1 -13287.727,E2 -13287.727} C_VEL
LIN {X 0,Y 357.888,Z 245.86,A -85,B 0,C 180,E1 -13288.478,E2 -13288.478} C_VEL
LIN {X 0,Y 358.323,Z 240.206,A -85,B 0,C 180,E1 -13289.014,E2 -13289.014} C_VEL
LIN {X 0,Y 356.762,Z 230.571,A -85,B 0,C 180,E1 -13289.847,E2 -13289.847} C_VEL
LIN {X 0,Y 354.595,Z 221.256,A -85,B 0,C 180,E1 -13290.515,E2 -13290.515} C_VEL
LIN {X 0,Y 353.867,Z 217.979,A -85,B 0,C 180,E1 -13290.725,E2 -13290.725} C_VEL
LIN {X 0,Y 354.023,Z 213.844,A -85,B 0,C 180,E1 -13294.105,E2 -13294.105} C_VEL
LIN {X 0,Y 354.322,Z 209.373,A -85,B 0,C 180,E1 -13297.862,E2 -13297.862} C_VEL
LIN {X 0,Y 354.621,Z 205.139,A -85,B 0,C 180,E1 -13301.514,E2 -13301.514} C_VEL
LIN {X 0,Y 354.909,Z 201.146,A -85,B 0,C 180,E1 -13305.084,E2 -13305.084} C_VEL
LIN {X 0,Y 354.998,Z 198.638,A -85,B 0,C 180,E1 -13307.423,E2 -13307.423} C_VEL
LIN {X 0,Y 354.928,Z 197.448,A -85,B 0,C 180,E1 -13308.58,E2 -13308.58} C_VEL
LIN {X 0,Y 355.01,Z 197.08,A -85,B 0,C 180,E1 -13310.889,E2 -13310.889} C_VEL
LIN {X 0,Y 355.14,Z 197.067,A -85,B 0,C 180,E1 -13313.182,E2 -13313.182} C_VEL
LIN {X 0,Y 355.245,Z 197.049,A -85,B 0,C 180,E1 -13317.733,E2 -13317.733} C_VEL
LIN {X 0,Y 355.399,Z 197.029,A -85,B 0,C 180,E1 -13320.001,E2 -13320.001} C_VEL
LIN {X 0,Y 355.245,Z 197.049,A -85,B 0,C 180,E1 -13322.269,E2 -13322.269} C_VEL
LIN {X 0,Y 355.116,Z 197.065,A -85,B 0,C 180,E1 -13326.821,E2 -13326.821} C_VEL
LIN {X 0,Y 354.958,Z 197.084,A -85,B 0,C 180,E1 -13330.266,E2 -13330.266} C_VEL
LIN {X 0,Y 354.945,Z 197.086,A -85,B 0,C 180,E1 -13334.02,E2 -13334.02} C_VEL
LIN {X 0,Y 354.925,Z 197.088,A -85,B 0,C 180,E1 -13338.109,E2 -13338.109} C_VEL
LIN {X 0,Y 354.837,Z 197.099,A -85,B 0,C 180,E1 -13342.107,E2 -13342.107} C_VEL
LIN {X 0,Y 354.901,Z 197.088,A -85,B 0,C 180,E1 -13345.828,E2 -13345.828} C_VEL
LIN {X 0,Y 354.856,Z 197.097,A -85,B 0,C 180,E1 -13349.679,E2 -13349.679} C_VEL
LIN {X 0,Y 354.808,Z 197.101,A -85,B 0,C 180,E1 -13353.703,E2 -13353.703} C_VEL
LIN {X 0,Y 354.8,Z 197.103,A -85,B 0,C 180,E1 -13356.46,E2 -13356.46} C_VEL
LIN {X 0,Y 354.826,Z 197.102,A -85,B 0,C 180,E1 -13359.424,E2 -13359.424} C_VEL
LIN {X 0,Y 354.79,Z 197.108,A -85,B 0,C 180,E1 -13362.868,E2 -13362.868} C_VEL
LIN {X 0,Y 354.769,Z 197.111,A -85,B 0,C 180,E1 -13366.104,E2 -13366.104} C_VEL
LIN {X 0,Y 354.829,Z 197.204,A -85,B 0,C 180,E1 -13369.454,E2 -13369.454} C_VEL
LIN {X 0,Y 355.6,Z 201.13,A -85,B 0,C 180,E1 -13372.238,E2 -13372.238} C_VEL
LIN {X 0,Y 356.637,Z 206.744,A -85,B 0,C 180,E1 -13375.861,E2 -13375.861} C_VEL
LIN {X 0,Y 357.1,Z 210.118,A -85,B 0,C 180,E1 -13377.901,E2 -13377.901} C_VEL
LIN {X 0,Y 356.573,Z 214.854,A -85,B 0,C 180,E1 -13380.479,E2 -13380.479} C_VEL
LIN {X 0,Y 355.59,Z 222.087,A -85,B 0,C 180,E1 -13384.227,E2 -13384.227} C_VEL
LIN {X 0,Y 354.793,Z 229.463,A -85,B 0,C 180,E1 -13387.891,E2 -13387.891} C_VEL
LIN {X 0,Y 354.166,Z 236.986,A -85,B 0,C 180,E1 -13391.488,E2 -13391.488} C_VEL
